# B&R Automation Studio project CombinedLinenSoiledA9KAN (part 7)

#### can_stnCyclic.ab
```automation-basic
PROGRAM _CYCLIC
;----------------------------------------
;Version 1.00 08/02/2005 D.J. First Issue
;----------------------------------------

;The Category, Customer and values from TrackView database are only written every 20 seconds
;unless the database has changed D[65] from TrackView
TimeNow  = clock_ms()
TimeDiff = UINT(TimeNow - TimeLastWrite)
IF (TimeDiff >= 20000) THEN
	WriteEvent 		= TRUE
	TimeLastWrite 	= TimeNow
ELSE IF D[65] <> DatabaseChanged THEN
	WriteEvent 		= TRUE
	TimeLastWrite 	= TimeNow
	DatabaseChanged = D[65]
ENDIF

IF CANOK THEN

	;----------------
	;Set Write values
	;----------------

	;Suction Box 1
	IF Box[1].BagReady THEN
		WriteFrame1021.ControlSignals = BIT_SET(WriteFrame1021.ControlSignals, 1)
	ELSE
		WriteFrame1021.ControlSignals = BIT_CLR(WriteFrame1021.ControlSignals, 1)
	ENDIF

	WriteFrame1101.SP1			= Box[1].SP1
	WriteFrame1101.SP2			= Box[1].SP2
	WriteFrame1101.SP3			= Box[1].SP3
	WriteFrame1101.Category 	= UINT(Box[1].Category)

	WriteFrame1111.Customer 	= Box[1].Customer
	WriteFrame1111.Destination 	= USINT(Box[1].Destination)

	EventWrite1021 = TRUE
	EventWrite1101 = WriteEvent
	EventWrite1111 = WriteEvent
	;Suction Box 1

	;Suction Box 2
	IF Box[2].BagReady THEN
		WriteFrame1022.ControlSignals = BIT_SET(WriteFrame1022.ControlSignals, 1)
	ELSE
		WriteFrame1022.ControlSignals = BIT_CLR(WriteFrame1022.ControlSignals, 1)
	ENDIF

	WriteFrame1102.SP1			= Box[2].SP1
	WriteFrame1102.SP2			= Box[2].SP2
	WriteFrame1102.SP3			= Box[2].SP3
	WriteFrame1102.Category 	= UINT(Box[2].Category)

	WriteFrame1112.Customer 	= Box[2].Customer
	WriteFrame1112.Destination 	= USINT(Box[2].Destination)

	EventWrite1022 = TRUE
	EventWrite1102 = WriteEvent
	EventWrite1112 = WriteEvent
	;Suction Box 2

	;Suction Box 3
	IF Box[3].BagReady THEN
		WriteFrame1023.ControlSignals = BIT_SET(WriteFrame1023.ControlSignals, 1)
	ELSE
		WriteFrame1023.ControlSignals = BIT_CLR(WriteFrame1023.ControlSignals, 1)
	ENDIF

	WriteFrame1103.SP1			= Box[3].SP1
	WriteFrame1103.SP2			= Box[3].SP2
	WriteFrame1103.SP3			= Box[3].SP3
	WriteFrame1103.Category 	= UINT(Box[3].Category)

	WriteFrame1113.Customer 	= Box[3].Customer
	WriteFrame1113.Destination 	= USINT(Box[3].Destination)

	EventWrite1023 = TRUE
	EventWrite1103 = WriteEvent
	EventWrite1113 = WriteEvent
	;Suction Box 3

	;Suction Box 4
	IF Box[4].BagReady THEN
		WriteFrame1024.ControlSignals = BIT_SET(WriteFrame1024.ControlSignals, 1)
	ELSE
		WriteFrame1024.ControlSignals = BIT_CLR(WriteFrame1024.ControlSignals, 1)
	ENDIF

	WriteFrame1104.SP1			= Box[4].SP1
	WriteFrame1104.SP2			= Box[4].SP2
	WriteFrame1104.SP3			= Box[4].SP3
	WriteFrame1104.Category 	= UINT(Box[4].Category)

	WriteFrame1114.Customer 	= Box[4].Customer
	WriteFrame1114.Destination 	= USINT(Box[4].Destination)

	EventWrite1024 = TRUE
	EventWrite1104 = WriteEvent
	EventWrite1114 = WriteEvent
	;Suction Box 4

	;Suction Box 5
	IF Box[5].BagReady THEN
		WriteFrame1025.ControlSignals = BIT_SET(WriteFrame1025.ControlSignals, 1)
	ELSE
		WriteFrame1025.ControlSignals = BIT_CLR(WriteFrame1025.ControlSignals, 1)
	ENDIF

	WriteFrame1105.SP1			= Box[5].SP1
	WriteFrame1105.SP2			= Box[5].SP2
	WriteFrame1105.SP3			= Box[5].SP3
	WriteFrame1105.Category 	= UINT(Box[5].Category)

	WriteFrame1115.Customer 	= Box[5].Customer
	WriteFrame1115.Destination 	= USINT(Box[5].Destination)

	EventWrite1025 = TRUE
	EventWrite1105 = WriteEvent
	EventWrite1115 = WriteEvent
	;Suction Box 5

	;Suction Box 6
	IF Box[6].BagReady THEN
		WriteFrame1026.ControlSignals = BIT_SET(WriteFrame1026.ControlSignals, 1)
	ELSE
		WriteFrame1026.ControlSignals = BIT_CLR(WriteFrame1026.ControlSignals, 1)
	ENDIF

	WriteFrame1106.SP1			= Box[6].SP1
	WriteFrame1106.SP2			= Box[6].SP2
	WriteFrame1106.SP3			= Box[6].SP3
	WriteFrame1106.Category 	= UINT(Box[6].Category)

	WriteFrame1116.Customer 	= Box[6].Customer
	WriteFrame1116.Destination 	= USINT(Box[6].Destination)

	EventWrite1026 = TRUE
	EventWrite1106 = WriteEvent
	EventWrite1116 = WriteEvent
	;Suction Box 6

	;Suction Box 7
	IF Box[7].BagReady THEN
		WriteFrame1027.ControlSignals = BIT_SET(WriteFrame1027.ControlSignals, 1)
	ELSE
		WriteFrame1027.ControlSignals = BIT_CLR(WriteFrame1027.ControlSignals, 1)
	ENDIF

	WriteFrame1107.SP1			= Box[7].SP1
	WriteFrame1107.SP2			= Box[7].SP2
	WriteFrame1107.SP3			= Box[7].SP3
	WriteFrame1107.Category 	= UINT(Box[7].Category)

	WriteFrame1117.Customer 	= Box[7].Customer
	WriteFrame1117.Destination 	= USINT(Box[7].Destination)

	EventWrite1027 = TRUE
	EventWrite1107 = WriteEvent
	EventWrite1117 = WriteEvent
	;Suction Box 7

	;Suction Box 8
	IF Box[8].BagReady THEN
		WriteFrame1028.ControlSignals = BIT_SET(WriteFrame1028.ControlSignals, 1)
	ELSE
		WriteFrame1028.ControlSignals = BIT_CLR(WriteFrame1028.ControlSignals, 1)
	ENDIF

	WriteFrame1108.SP1			= Box[8].SP1
	WriteFrame1108.SP2			= Box[8].SP2
	WriteFrame1108.SP3			= Box[8].SP3
	WriteFrame1108.Category 	= UINT(Box[8].Category)

	WriteFrame1118.Customer 	= Box[8].Customer
	WriteFrame1118.Destination 	= USINT(Box[8].Destination)

	EventWrite1028 = TRUE
	EventWrite1108 = WriteEvent
	EventWrite1118 = WriteEvent
	;Suction Box 8

	;Suction Box 9
	IF Box[9].BagReady THEN
		WriteFrame1029.ControlSignals = BIT_SET(WriteFrame1029.ControlSignals, 1)
	ELSE
		WriteFrame1029.ControlSignals = BIT_CLR(WriteFrame1029.ControlSignals, 1)
	ENDIF

	WriteFrame1109.SP1			= Box[9].SP1
	WriteFrame1109.SP2			= Box[9].SP2
	WriteFrame1109.SP3			= Box[9].SP3
	WriteFrame1109.Category 	= UINT(Box[9].Category)

	WriteFrame1119.Customer 	= Box[9].Customer
	WriteFrame1119.Destination 	= USINT(Box[9].Destination)

	EventWrite1029 = TRUE
	EventWrite1109 = WriteEvent
	EventWrite1119 = WriteEvent
	;Suction Box 9

	;-----------------
	;Service CAN table
	;-----------------

	IF CANdftab_01.status=0 THEN						(*check error level*)
		CANrwtab_01.enable		= 1
		CANrwtab_01.tab_ident	= CANdftab_01.tab_ident (*define tab_id*)
		CANrwtab_01 FUB CANrwtab()						(*initiate CANrwtab*)
		LastError = CANrwtab_01.status
	ENDIF

	;----------------------------------
	;Check for incomming data from CBW1
	;----------------------------------

	;Box 1
	IF EventRead1001 THEN
		EventRead1001 = FALSE
		Box1Cus = UINT(ReadFrame1001.Customer)
	ENDIF

	IF EventRead1011 THEN

		EventRead1011 = FALSE

		Box[1].Live 		= BIT_TST(ReadFrame1011.ControlSignals,0)
		Box[1].LoadFinished = BIT_TST(ReadFrame1011.ControlSignals,1)

		Box[1].Weight		= ReadFrame1011.Weight
		IF (Box1Cus > 0) THEN
			Bag[201].Cus = Box1Cus
		ENDIF
		IF Box[1].Live THEN
			Box[1].LiveTime = 50	;5 seconds
		ENDIF

	ENDIF

;	IF EDGEPOS (Box[1].LoadFinished = 0) THEN
;		Bag[201].Cus = Box1Cus
;	ENDIF
;
;	IF (Bag[201].Cus = 0) THEN
;		Bag[201].Cus = Box1Cus
;	ENDIF

	;Box 2
	IF EventRead1002 THEN
		EventRead1002 = FALSE
		Box2Cus = UINT(ReadFrame1002.Customer)
	ENDIF

	IF EventRead1012 THEN

		EventRead1012 = FALSE

		Box[2].Live 		= BIT_TST(ReadFrame1012.ControlSignals,0)
		Box[2].LoadFinished = BIT_TST(ReadFrame1012.ControlSignals,1)

		Box[2].Weight		= ReadFrame1012.Weight
		IF (Box2Cus > 0) THEN
			Bag[202].Cus = Box2Cus
		ENDIF
		IF Box[2].Live THEN
			Box[2].LiveTime = 50	;5 seconds
		ENDIF

	ENDIF

;	IF EDGEPOS (Box[2].LoadFinished = 0) THEN
;		Bag[202].Cus = Box2Cus
;	ENDIF
;
;	IF (Bag[202].Cus = 0) THEN
;		Bag[202].Cus = Box2Cus
;	ENDIF

	;Box 3
	IF EventRead1003 THEN
		EventRead1003 = FALSE
		Box3Cus = UINT(ReadFrame1003.Customer)
	ENDIF

	IF EventRead1013 THEN

		EventRead1013 = FALSE

		Box[3].Live 		= BIT_TST(ReadFrame1013.ControlSignals,0)
		Box[3].LoadFinished = BIT_TST(ReadFrame1013.ControlSignals,1)

		Box[3].Weight		= ReadFrame1013.Weight
		IF (Box3Cus > 0) THEN
				Bag[203].Cus = Box3Cus
		ENDIF
		IF Box[3].Live THEN
			Box[3].LiveTime = 50	;5 seconds
		ENDIF

	ENDIF

;	IF EDGEPOS (Box[3].LoadFinished = 0) THEN
;		Bag[203].Cus = Box3Cus
;	ENDIF
;
;	IF (Bag[203].Cus = 0) THEN
;		Bag[203].Cus = Box3Cus
;	ENDIF

	;Box 4
	IF EventRead1004 THEN
		EventRead1004 = FALSE
		Box4Cus = UINT(ReadFrame1004.Customer)
	ENDIF

	IF EventRead1014 THEN

		EventRead1014 = FALSE

		Box[4].Live 		= BIT_TST(ReadFrame1014.ControlSignals,0)
		Box[4].LoadFinished = BIT_TST(ReadFrame1014.ControlSignals,1)

		Box[4].Weight		= ReadFrame1014.Weight
		IF (Box4Cus > 0) THEN
			Bag[204].Cus = Box4Cus
		ENDIF
		IF Box[4].Live THEN
			Box[4].LiveTime = 50	;5 seconds
		ENDIF

	ENDIF

;	IF EDGEPOS (Box[4].LoadFinished = 0) THEN
;		Bag[204].Cus = Box4Cus
;	ENDIF
;
;	IF (Bag[204].Cus = 0) THEN
;		Bag[204].Cus = Box4Cus
;	ENDIF

	;Box 5
	IF EventRead1005 THEN
		EventRead1005 = FALSE
		Box5Cus = UINT(ReadFrame1005.Customer)
	ENDIF

	IF EventRead1015 THEN

		EventRead1015 = FALSE

		Box[5].Live 		= BIT_TST(ReadFrame1015.ControlSignals,0)
		Box[5].LoadFinished = BIT_TST(ReadFrame1015.ControlSignals,1)

			Box[5].Weight		= ReadFrame1015.Weight
		IF (Box5Cus > 0) THEN
			Bag[205].Cus = Box5Cus
		ENDIF
		IF Box[5].Live THEN
			Box[5].LiveTime = 50	;5 seconds
		ENDIF

	ENDIF

;	IF EDGEPOS (Box[5].LoadFinished = 0) THEN
;		Bag[205].Cus = Box5Cus
;	ENDIF
;
;	IF (Bag[205].Cus = 0) THEN
;		Bag[205].Cus = Box5Cus
;	ENDIF

	;Box 6
	IF EventRead1006 THEN
		EventRead1006 = FALSE
		Box6Cus = UINT(ReadFrame1006.Customer)
	ENDIF

	IF EventRead1016 THEN

		EventRead1016 = FALSE

		Box[6].Live 		= BIT_TST(ReadFrame1016.ControlSignals,0)
		Box[6].LoadFinished = BIT_TST(ReadFrame1016.ControlSignals,1)

		Box[6].Weight		= ReadFrame1016.Weight
		IF (Box6Cus > 0) THEN
			Bag[206].Cus = Box6Cus
		ENDIF
		IF Box[6].Live THEN
			Box[6].LiveTime = 50	;5 seconds
		ENDIF

	ENDIF

;	IF EDGEPOS (Box[6].LoadFinished = 0) THEN
;		Bag[206].Cus = Box6Cus
;	ENDIF
;
;	IF (Bag[206].Cus = 0) THEN
;		Bag[206].Cus = Box6Cus
;	ENDIF

	;Box 7
	IF EventRead1007 THEN
		EventRead1007 = FALSE
		Dummy = ReadFrame1007.Customer
	ENDIF

	IF EventRead1017 THEN

		EventRead1017 = FALSE

		Box[7].Live 		= BIT_TST(ReadFrame1017.ControlSignals,0)
		Box[7].LoadFinished = BIT_TST(ReadFrame1017.ControlSignals,1)

		Box[7].Weight		= ReadFrame1017.Weight
			IF (ReadFrame1007.Customer > 0) THEN
				Bag[207].Cus = ReadFrame1007.Customer
			ENDIF
		IF Box[7].Live THEN
			Box[7].LiveTime = 50	;5 seconds
		ENDIF

	ENDIF

	;Box 8
	IF EventRead1008 THEN
		EventRead1008 = FALSE
		Dummy = ReadFrame1008.Customer
	ENDIF

	IF EventRead1018 THEN

		EventRead1018 = FALSE

		Box[8].Live 		= BIT_TST(ReadFrame1018.ControlSignals,0)
		Box[8].LoadFinished = BIT_TST(ReadFrame1018.ControlSignals,1)

		Box[8].Weight		= ReadFrame1018.Weight
			IF (ReadFrame1008.Customer > 0) THEN
				Bag[208].Cus = ReadFrame1008.Customer
			ENDIF
		IF Box[8].Live THEN
			Box[8].LiveTime = 50	;5 seconds
		ENDIF

	ENDIF

	;Box 9
	IF EventRead1009 THEN
		EventRead1009 = FALSE
		Dummy = ReadFrame1009.Customer
	ENDIF

	IF EventRead1019 THEN

		EventRead1019 = FALSE

		Box[9].Live 		= BIT_TST(ReadFrame1019.ControlSignals,0)
		Box[9].LoadFinished = BIT_TST(ReadFrame1019.ControlSignals,1)
			Box[9].ReadyToLoad = BIT_TST(ReadFrame1019.ControlSignals,2)
			Box[9].Weight		= ReadFrame1019.Weight
			IF (ReadFrame1009.Customer > 0) THEN
				Bag[209].Cus = ReadFrame1009.Customer
			ENDIF
		IF Box[9].Live THEN
			Box[9].LiveTime = 50	;5 seconds
		ENDIF

	ENDIF

	;-------------------
	;CAN Live / Presence
	;-------------------

	LOOP n = 1 TO 9 DO

		IF (Box[n].LiveTime > 0) THEN
			Box[n].LiveTime = (Box[n].LiveTime - 1)
		ENDIF

		Box[n].Live = (Box[n].LiveTime <> 0)

	ENDLOOP

ENDIF

;Reset Write Event - 20 seconds or Event
WriteEvent = FALSE
END_PROGRAM
```

#### can_stnInit.ab
```automation-basic
PROGRAM _INIT
	(* init program *)

CAN_enable = 1

;BOX 1 Reset CAN data table READ and WRITE events
EventRead1001 	= 0
EventRead1011 	= 0
EventWrite1021 	= 0
EventWrite1101 	= 0
EventWrite1111 	= 0

;BOX 2 Reset CAN data table READ and WRITE events
EventRead1002 	= 0
EventRead1012 	= 0
EventWrite1022 	= 0
EventWrite1102 	= 0
EventWrite1112 	= 0

;BOX 3 Reset CAN data table READ and WRITE events
EventRead1003 	= 0
EventRead1013 	= 0
EventWrite1023 	= 0
EventWrite1103 	= 0
EventWrite1113 	= 0

;BOX 4 Reset CAN data table READ and WRITE events
EventRead1004 	= 0
EventRead1014 	= 0
EventWrite1024 	= 0
EventWrite1104 	= 0
EventWrite1114 	= 0

;BOX 5 Reset CAN data table READ and WRITE events
EventRead1005 	= 0
EventRead1015 	= 0
EventWrite1025 	= 0
EventWrite1105 	= 0
EventWrite1115 	= 0

;BOX 6 Reset CAN data table READ and WRITE events
EventRead1006 	= 0
EventRead1016 	= 0
EventWrite1026 	= 0
EventWrite1106 	= 0
EventWrite1116 	= 0

;BOX 7 Reset CAN data table READ and WRITE events
EventRead1007 	= 0
EventRead1017 	= 0
EventWrite1027 	= 0
EventWrite1107 	= 0
EventWrite1117 	= 0

;BOX 8 Reset CAN data table READ and WRITE events
EventRead1008 	= 0
EventRead1018 	= 0
EventWrite1028 	= 0
EventWrite1108 	= 0
EventWrite1118 	= 0

;BOX 9 Reset CAN data table READ and WRITE events
EventRead1009 	= 0
EventRead1019 	= 0
EventWrite1029 	= 0
EventWrite1109 	= 0
EventWrite1119 	= 0

strcpy(ADR(strName_can_tab), "can_stns")
DOInfo.enable = TRUE
DOInfo.pName  = ADR(strName_can_tab)
DOInfo FUB DatObjInfo()

wTabNum 				= WORD(DOInfo.len / 72)	;Define number of values

CANopen_01.enable		= CAN_enable
CANopen_01.baud_rate	= 25					;Define baud rate - 250 kbit/s
CANopen_01.cob_anz		= wTabNum      			;Define number of link objects
CANopen_01.error_adr	= ADR(error_var)		;Define address for error output
CANopen_01.device		= ADR("SS1.IF1")	    ;Define number of device
CANopen_01.info			= 0

CANopen_01 FUB CANopen()						;Initiate CANopen

IF CANopen_01.status = 0 THEN					;Check error level

	IF (DOInfo.status = 0) THEN

		CANdftab_01.enable			= TRUE
		CANdftab_01.us_ident 		= CANopen_01.us_ident	;Set us_id
		CANdftab_01.table_adr		= DOInfo.pDatObjMem		;Define address of data object
		CANdftab_01.tab_num			= wTabNum

		CANdftab_01 FUB CANdftab()    						;Initiate CANdftab

		IF CANdftab_01.status = 0 THEN
			WriteFrame1021.ControlSignals = BIT_SET(WriteFrame1021.ControlSignals,0);Set Live Signal
			WriteFrame1022.ControlSignals = BIT_SET(WriteFrame1022.ControlSignals,0)
			WriteFrame1023.ControlSignals = BIT_SET(WriteFrame1023.ControlSignals,0)
			WriteFrame1024.ControlSignals = BIT_SET(WriteFrame1024.ControlSignals,0);Set Live Signal
			WriteFrame1025.ControlSignals = BIT_SET(WriteFrame1025.ControlSignals,0)
			WriteFrame1026.ControlSignals = BIT_SET(WriteFrame1026.ControlSignals,0)
			WriteFrame1027.ControlSignals = BIT_SET(WriteFrame1027.ControlSignals,0);Set Live Signal
			WriteFrame1028.ControlSignals = BIT_SET(WriteFrame1028.ControlSignals,0)
			WriteFrame1029.ControlSignals = BIT_SET(WriteFrame1029.ControlSignals,0)
			CANOK = TRUE
		ENDIF

	ENDIF

ENDIF
END_PROGRAM
```

- Data object Logical/Mewa/200ms/CAN/can_stns (Simple, version 1.00.0) - * Suction system (no source held here)

### Program Logical/Mewa/200ms/CAN/can_live (IEC) - * CAN Live status 1-32 to TrackView

#### can_live.ab
```automation-basic
PROGRAM _CYCLIC
(* cyclic program *)

;------------------------------------------
;CAN Live / Status indication to TrackView
;------------------------------------------

;-----------------------------------------
;Revision 1.00 24/11/2005 D.J. First Issue
;-----------------------------------------

;Move CAN Status to Registers

;1-16
CANLive_1.Input[0] = CAN[1].Live
CANLive_1.Input[1] = CAN[2].Live
CANLive_1.Input[2] = CAN[3].Live
CANLive_1.Input[3] = CAN[4].Live
CANLive_1.Input[4] = CAN[5].Live
CANLive_1.Input[5] = CAN[6].Live
CANLive_1.Input[6] = CAN[7].Live
CANLive_1.Input[7] = CAN[8].Live
CANLive_1.Input[8] = CAN[9].Live
CANLive_1.Input[9] = CAN[10].Live
CANLive_1.Input[10] = FALSE ;Box[1].Live
CANLive_1.Input[11] = FALSE ;Box[2].Live
CANLive_1.Input[12] = FALSE ;Box[3].Live
CANLive_1.Input[13] = FALSE ;Box[4].Live
CANLive_1.Input[14] = FALSE ;Box[5].Live
CANLive_1.Input[15] = FALSE ;Box[6].Live

CANLive_1 FUB BIT_ENCODE()

D[76] = CANLive_1.Output

;17-32
CANLive_2.Input[0] = FALSE ;Box[7].Live
CANLive_2.Input[1] = FALSE ;Box[8].Live
CANLive_2.Input[2] = FALSE ;Box[9].Live
CANLive_2.Input[3] = CAN[20].Live
CANLive_2.Input[4] = CAN[21].Live
CANLive_2.Input[5] = CAN[22].Live
CANLive_2.Input[6] = CAN[23].Live
CANLive_2.Input[7] = CAN[24].Live
CANLive_2.Input[8] = CAN[25].Live
CANLive_2.Input[9] = CAN[26].Live
CANLive_2.Input[10] = CAN[27].Live
CANLive_2.Input[11] = CAN[28].Live
CANLive_2.Input[12] = CAN[29].Live
CANLive_2.Input[13] = CAN[30].Live
CANLive_2.Input[14] = CAN[31].Live
CANLive_2.Input[15] = CAN[32].Live

CANLive_2 FUB BIT_ENCODE()

D[77] = CANLive_2.Output
END_PROGRAM
```

### Package Logical/Mewa/KanLink - KanLink Setup tasks

### KanLink.typ - Global data types
```iecst
(********************************************************************
 * COPYRIGHT -- HP
 ********************************************************************
 * Package: KanLink
 * File: KanLink.typ
 * Author: treamsbottom
 * Created: April 23, 2012
 ********************************************************************
 * Data types of package KanLink
 ********************************************************************)

TYPE
	State_typ : 	STRUCT
		Estop : USINT := 1;
		Fault : USINT := 3;
		OK : USINT := 6;
		Warning : USINT := 10;
	END_STRUCT;
	KanLink_Param_typ : 	STRUCT
		Mcn_no : UINT;
		Area : UINT;
		Adr : UINT;
	END_STRUCT;
END_TYPE
```

### KanLink.var - Global variables
```iecst
(********************************************************************
 * COPYRIGHT -- HP
 ********************************************************************
 * Package: KanLink
 * File: KanLink.var
 * Author: treamsbottom
 * Created: April 23, 2012
 ********************************************************************
 * Variables of package KanLink
 ********************************************************************)
VAR
	Batch : ARRAY[0..9] OF BatchData_typ;
	Kan : ARRAY[0..9] OF BatchData_typ;
	PTResp : ARRAY[0..9] OF KL_BTxf_typ;
	PT100 : ARRAY[0..9] OF KL_BTxf_typ;
	McState : State_typ;
END_VAR
VAR RETAIN
	KanLink_Param : ARRAY[0..9] OF KanLink_Param_typ;
END_VAR
```

### Program Logical/Mewa/KanLink/Kan_Drv (IEC) - Empty base sequence

#### Kan_Drv.ab
```automation-basic
;--------------------------------------------
;Sequence Kan_Drv
;--------------------------------------------

PROGRAM _INIT
(* init program *)
END_PROGRAM

PROGRAM _CYCLIC

// Batch Transfer Handshake
//Please enter the index of Kan Bag you want to transfer to the PT+ This was set up in BatchInfo.task
LOOP n = 0 TO (Std.MaxKanLink) DO
;LOOP n = 0 TO 1 DO
	PT100[n].Resp.BatchData = Kan[n];

	ValidCat = 	strcmp(ADR(CAN[n+1].Category), "")
	IF (ValidCat <> 0)THEN
			PT100[n].Resp.xHsDataValid = TRUE;
	ELSE
		PT100[n].Resp.xHsDataValid = FALSE
		PT100[n].Resp.xHsUnloading = FALSE
	ENDIF

	IF CAN[n+1].BagReady THEN
		PT100[n].Resp.xHsReqForUnload = TRUE;
	ELSE
		PT100[n].Resp.xHsReqForUnload = FALSE;
	ENDIF

	CAN[n+1].DropLoad 		= PT100[n].Req.xHreadyForLoad;
	CAN[n+1].LoadDropped  	= PT100[n].Req.xHbatchReceived;
	;CAN[n].Live				= Kanl

		IF CAN[n+1].DropLoad THEN
		PT100[n].Resp.xHsUnloading = TRUE
	ENDIF

	CAN[n+1].Live = IFhlKanLink.Server[n].out.xConnected
	;Status Feedback
	IF Std.HaltSys THEN
		PT100[n].Resp.wState = McState.Estop
	ELSE IF (D[200] > 0) THEN ; alarm present
		PT100[n].Resp.wState = McState.Fault
	ELSE
		PT100[n].Resp.wState = McState.OK
	ENDIF
ENDLOOP
END_PROGRAM
```

#### Kan_Drv.var
```iecst
VAR
	n : UINT;
	ValidCat : DINT;
END_VAR
```

### Program Logical/Mewa/KanLink/zzKanLink (IEC) - KanLink Set up

#### zzKanLinkCyclic.ab - Cyclic code
```automation-basic
(********************************************************************
 * COPYRIGHT -- HP
 ********************************************************************
 * Program: zzKanLink
 * File: zzKanLinkCyclic.ab
 * Author: treamsbottom
 * Created: April 23, 2012
 ********************************************************************
 * Implementation of program zzKanLink
 ********************************************************************)

PROGRAM _CYCLIC
IF NOT init THEN
	KanLink_Param[0].Adr = 12
	KanLink_Param[0].Area = 3
	KanLink_Param[1].Adr = 11
	KanLink_Param[1].Area = 3
	LOOP n = 0 TO (Std.MaxKanLink) DO
	;LOOP n = 0 TO 2 DO
	;Build strings to pass to variable names, only required in a loop as index number changes.
		itoa(n,ADR(sn))	; put n into string
		strcpy(ADR(sReq),"PT100[");build string for variable name (request)
		strcat(ADR(sReq),ADR(sn))
		strcat(ADR(sReq),"].Req")
		strcpy(ADR(sResp),"PT100[");;build string for variable name (response)
		strcat(ADR(sResp),ADR(sn))
		strcat(ADR(sResp),"].Resp")

		IFhlKanLink.Parameter.Server[n].Adr = KanLink_Param[n].Adr ; Populate these arrays .
		IFhlKanLink.Parameter.Server[n].Area = KanLink_Param[n].Area
		IFhlKanLink.Parameter.Server[n].Cmd = 1000 ; cmd from the server are always even
		IFhlKanLink.Parameter.Server[n].CmdOpt = 0
		IFhlKanLink.Parameter.Server[n].TimeOut = 1000 ;ms
		strcpy(ADR(IFhlKanLink.Parameter.Server[n].Name),"PT100") ; Diags Only
		strcpy(ADR(IFhlKanLink.Parameter.Server[n].sReq),ADR(sReq));"zzKanLink:PT100[0].Req")
		strcpy(ADR(IFhlKanLink.Parameter.Server[n].sResp),ADR(sResp));"zzKanLink:PT100[0].Resp")
	ENDLOOP

	;Clean side- Only 1 client for talking to shuttle/driers can be put into a loop as the soiled.
;	IFhlKanLink.Parameter.Client[0].Adr = 15
;	IFhlKanLink.Parameter.Client[0].Area = 3
;	IFhlKanLink.Parameter.Client[0].Cmd = 1000
;	IFhlKanLink.Parameter.Client[0].CmdOpt = 0
;	IFhlKanLink.Parameter.Client[0].CycleTime = 1000;ms
;	strcpy(ADR(IFhlKanLink.Parameter.Client[0].Name),"PTResp")
;	strcpy(ADR(IFhlKanLink.Parameter.Client[0].sReq),"PTResp[0].Req")
;	strcpy(ADR(IFhlKanLink.Parameter.Client[0].sResp),"PTResp[0].Resp")

	IFhlKanLink.in.xRestart = TRUE
	IFmnParam.Out.xParamOK = TRUE
	init = TRUE
	PT100 ; Variable that writes to the PT+
	PTResp ; Variable that reads from PT+ (Clean Side)
ENDIF

END_PROGRAM
```

#### zzKanLinkInit.ab - Initialization code
```automation-basic
(********************************************************************
 * COPYRIGHT -- HP
 ********************************************************************
 * Program: zzKanLink
 * File: zzKanLinkInit.ab
 * Author: treamsbottom
 * Created: April 23, 2012
 ********************************************************************
 * Implementation of program zzKanLink
 ********************************************************************)

PROGRAM _INIT

(* TODO : Add your code here *)

END_PROGRAM
```

#### zzKanLink.var - Local variables
```iecst
(********************************************************************
 * COPYRIGHT -- HP
 ********************************************************************
 * Program: zzKanLink
 * File: zzKanLink.var
 * Author: treamsbottom
 * Created: April 23, 2012
 ********************************************************************
 * Local variables of program zzKanLink
 ********************************************************************)
VAR
	init : BOOL;
	n : UINT;
	sReq : STRING[80];
	sn : STRING[2];
	sResp : STRING[80];
END_VAR
```

### Program Logical/Mewa/KanLink/BatchInfo (IEC) - Empty base sequence

#### BatchInfo.ab
```automation-basic
;--------------------------------------------
;Sequence BatchInfo
;--------------------------------------------

PROGRAM _INIT
(* init program *)
END_PROGRAM

PROGRAM _CYCLIC

	;Please enter Bag number to to send via KannLink Batch info (1002)
	BagNum[0]	= 55
	BagNum[1]	= 60
	BagNum[2]	= 0
	BagNum[3]	= 0
	BagNum[4]	= 0
	BagNum[5]	= 0

	LOOP n = 0 TO Std.MaxKanLink DO
		IF Bag[BagNum[n]].Cat > 0 THEN
			GetTimeStamp.enable = 1
			GetTimeStamp FUB DTGetTime()
			Kan[n].dtTimeStamp = GetTimeStamp.DT1

			;Make a string out of CAT and CUS
			length := itoa(Bag[BagNum[n]].Cat,ADR(myCategoryString));
			length := itoa(Bag[BagNum[n]].Cus,ADR(myCustomerString));
			;strcpy(ADR(myCategoryString),ADR(Bag[BagNum[n]].Cat))
			;strcpy(ADR(myCustomerString),ADR(Bag[BagNum[n]].Cus))

			;copy Bag Data to KanLink Bag data type
			Kan[n].bCntCustomers = 1
			Kan[n].sCategory = myCategoryString
			Kan[n].wTotalWeight = Bag[BagNum[n]].Wgt ;Summaray weight of all Part Customers in the Bag, normally 1
			;Frist Customer in the Bag, allowed for multible Customers in future
			Kan[n].PartBatch[0].sCustomNo = myCustomerString
			Kan[n].PartBatch[0].wCustomWeight = Bag[BagNum[n]].Wgt
		ELSE
			strcpy(ADR(myCategoryString),ADR(""));
			strcpy(ADR(myCustomerString),ADR(""));
			Kan[n].bCntCustomers = 0
			Kan[n].sCategory = myCategoryString
			Kan[n].wTotalWeight = 0 ;Summaray weight of all Part Customers in the Bag, normally 1
			;Frist Customer in the Bag, allowed for multible Customers in future
			Kan[n].PartBatch[0].sCustomNo = myCustomerString
			Kan[n].PartBatch[0].wCustomWeight = 0
		ENDIF
		Batch[n] = Kan[n] ; Populate array for PT+ PVI
	ENDLOOP
;
;	//Batch info for all Batches
;	Bel_1_BI.Resp.BatchData[0] = Kan[0];
;	Bel_1_BI.Resp.BatchData[1] = Kan[0];
;	Bel_1_BI.Resp.BatchData[2] = Kan[0];
;	Bel_1_BI.Resp.BatchData[3] = Kan[0];
;	Bel_1_BI.Resp.BatchData[4] = Kan[0];
;	Bel_1_BI.Resp.BatchData[5] = Kan[0];
;
;
;	IF (Bel_1_BI.Req.wCntPositions >= 0) THEN
;		n = Bel_1_BI.Req.wCntPositions;
;		Bel_1_BI.Resp.wCntPositions =  Bel_1_BI.Req.wCntPositions;
;		IF (n = 0) OR (n >= 1) THEN
;			Bel_1_BI.Resp.wNoOfPositions[0] = Bel_1_BI.Req.wNoOfPosition[0];
;			Bel_1_BI.Resp.BatchData[0] = Kan[Bel_1_BI.Req.wNoOfPosition[0]];
;		ENDIF
;		IF (n = 0) OR (n >= 2) THEN
;			Bel_1_BI.Resp.wNoOfPositions[1] = Bel_1_BI.Req.wNoOfPosition[1];
;			Bel_1_BI.Resp.BatchData[1] = Kan[Bel_1_BI.Req.wNoOfPosition[1]];
;		ENDIF
;		IF (n = 0) OR (n >= 3) THEN
;			Bel_1_BI.Resp.wNoOfPositions[2] = Bel_1_BI.Req.wNoOfPosition[2];
;			Bel_1_BI.Resp.BatchData[2] = Kan[Bel_1_BI.Req.wNoOfPosition[2]];
;		ENDIF
;		IF (n = 0) OR (n >= 4) THEN
;			Bel_1_BI.Resp.wNoOfPositions[3] = Bel_1_BI.Req.wNoOfPosition[3];
;			Bel_1_BI.Resp.BatchData[3] = Kan[Bel_1_BI.Req.wNoOfPosition[3]];
;		ENDIF
;		IF (n = 0) OR (n >= 5) THEN
;			Bel_1_BI.Resp.wNoOfPositions[4] = Bel_1_BI.Req.wNoOfPosition[4];
;			Bel_1_BI.Resp.BatchData[4] = Kan[Bel_1_BI.Req.wNoOfPosition[4]];
;		ENDIF
;		IF (n = 0) OR (n = 6) THEN
;			Bel_1_BI.Resp.wNoOfPositions[5] = Bel_1_BI.Req.wNoOfPosition[5];
;			Bel_1_BI.Resp.BatchData[5] = Kan[Bel_1_BI.Req.wNoOfPosition[5]];
;		ENDIF
;	ENDIF
;
;
;
END_PROGRAM
```

#### BatchInfo.var
```iecst
VAR
	BagNum : ARRAY[0..10] OF UINT;
	n : UINT;
	length : UINT;
	myCategoryString : STRING[11];
	myCustomerString : STRING[11];
	nxt_adr : UDINT;
	GetTimeStamp : DTGetTime;
END_VAR
```

### Package Logical/Mewa/KGFramework - Standard-Packages

### Package Logical/Mewa/KGFramework/Pkg_KGStandard - Kannegiesser Standards

### kgMachineState.var - Package variables
```iecst
(********************************************************************
 * COPYRIGHT -- Herbert Kannegiesser GmbH
 ********************************************************************
 * Package: Pkg_KGStandard
 * File: kgMachineState.var
 * Author: hunholz
 * Created: January 27, 2012
 ********************************************************************
 * Variables of package Pkg_KGStandard
 ********************************************************************)
VAR CONSTANT
	KG_MACHINESTATE_OFF : UINT := 0; (*Machine is turned off*)
	KG_MACHINESTATE_EMERGENCYSTOP : UINT := 1; (*Emergency stop*)
	KG_MACHINESTATE_SAFESTOP : UINT := 2; (*Safe stop*)
	KG_MACHINESTATE_FAULT : UINT := 3; (*Fault*)
	KG_MACHINESTATE_FAULT_GONE : UINT := 4; (*Fault, wait for acknowledge*)
	KG_MACHINESTATE_SERVICE : UINT := 5; (*Service*)
	KG_MACHINESTATE_AUTOMATIC_RUN : UINT := 6; (*Automatic Run*)
	KG_MACHINESTATE_STOP : UINT := 7; (*Stop*)
	KG_MACHINESTATE_WAIT_AUTOMATIC : UINT := 8; (*Automatic Wait (Standby)*)
	KG_MACHINESTATE_WAIT_MAN : UINT := 9; (*Automatic Wait for manual action*)
	KG_MACHINESTATE_WARNING : UINT := 10; (*Automatic Warning*)
END_VAR
(*Special states for dryer*)
VAR CONSTANT
	KG_MACHINESTATE_DRY_HEATING : UINT := 30; (*Automatic heating*)
	KG_MACHINESTATE_DRY_COOLDOWN : UINT := 31; (*Automatic cooldown*)
	KG_MACHINESTATE_DRY_CLEAN_FILTER : UINT := 32; (*Automatic clean filter*)
	KG_MACHINESTATE_DRY_AFTERRUN : UINT := 33; (*Automatic afterrun*)
	KG_MACHINESTATE_DRY_FAN_CLEAN : UINT := 34; (*Automatic running cleaning fan*)
END_VAR
(*Special states for conveyor*)
VAR CONSTANT
	KG_MACHINESTATE_CONV_FWD : UINT := 40; (*Automatic running forward*)
	KG_MACHINESTATE_CONV_FWD2 : UINT := 41; (*Automatic running forward 2nd speed*)
	KG_MACHINESTATE_CONV_REV : UINT := 42; (*Automatic running reverse*)
	KG_MACHINESTATE_CONV_REV2 : UINT := 43; (*Automatic running reverse 2nd speed*)
END_VAR
```

### Library Logical/Mewa/KGFramework/Pkg_KGStandard/KGstdLib (IEC) - Kannegiesser Hilfsfunktionen
Depends on: astime, AsIODiag, Ethernet, AsBrStr, DataObj, AsArLog

#### KGstdLib.var - Exported constants
```iecst
(********************************************************************
 * COPYRIGHT -- Microsoft
 ********************************************************************
 * Library: KGstd
 * File: KGstd.var
 * Author: hunholz
 * Created: June 23, 2011
 ********************************************************************
 * Constants of library KGstd
 ********************************************************************)
VAR CONSTANT
	KG_ERR_RB_NOREAD : UINT := 1;
	KG_ERR_RB_POINTER : UINT := 2;
	KG_ERR_RB_WRITEPOINTER : UINT := 3;
	KG_ERR_RB_READPOINTER : UINT := 4;
	KG_ERR_RB_STARTPOINTER : UINT := 5;
	KG_ERR_RB_LOCPOINTER : UINT := 6;
	KG_ERR_RB_SIZE : UINT := 7;
	KG_ERR_GETETHPORT_IFSTRING : UINT := 21;
	KG_ERR_GETETHPORT_ADRIF : UINT := 22;
	KG_ERR_WRONGSIZES : UINT := 30;
	KG_INFO_DO_NEW : UINT := 31;
	KG_ERR_NULPOINTER : UINT := 40;
	KG_ERR_NULLSTRING : UINT := 41;
END_VAR
(*RB Modus für kgRBloc*)
VAR CONSTANT
	KG_RB_LOC_MODE_ABSOLUTE : USINT := 0;
	KG_RB_LOC_MODE_FROMSTART : USINT := 1;
	KG_RB_LOC_MODE_FROMEND : USINT := 2;
END_VAR
(*CPU Identifier*)
VAR CONSTANT
	KG_CPU_X20CP3484 : UDINT := 16#23A6;
	KG_CPU_X20CP1484 : UDINT := 16#23A5;
	KG_CPU_X20CP1484_1 : UDINT := 16#AABE;
	KG_CPU_X20CP3484_1 : UDINT := 16#AABF;
	KG_CPU_X20CP1486 : UDINT := 16#2164;
	KG_CPU_X20CP3486 : UDINT := 16#1F19;
	KG_CPU_X20CP3585 : UDINT := 16#C3AF;
	KG_CPU_PP420_1043_75 : UDINT := 16#23BD;
	KG_CPU_PP65_0571_P74 : UDINT := 16#A964;
	KG_CPU_CTT_11 : UDINT := 16#A2BC;
	KG_CPU_PCT_03 : UDINT := 16#A7DD;
	KG_CPU_PCT_04 : UDINT := 16#B399;
END_VAR
(*Units*)
VAR CONSTANT
	KG_UNIT_METRIC : USINT := 0;
	KG_UNIT_US : USINT := 1;
END_VAR
```

#### KGstdLib.fun - Exported functions and function blocks
```iecst
(********************************************************************
 * COPYRIGHT -- Microsoft
 ********************************************************************
 * Library: KGstd
 * File: KGstd.fun
 * Author: hunholz
 * Created: June 23, 2011
 ********************************************************************
 * Functions and function blocks of library KGstd
 ********************************************************************)

FUNCTION_BLOCK kgGetEthPort (*Returns the CPUs ethernet port as string*)
	VAR_INPUT
		enable : BOOL;
		adrIF : UDINT;
	END_VAR
	VAR_OUTPUT
		status : UINT;
	END_VAR
	VAR
		_bStep : USINT;
		DiagCreateInfo_CPU : DiagCreateInfo;
		DiagGetNumInfo_CPU : DiagGetNumInfo;
		DiagDisposeInfo_CPU : DiagDisposeInfo;
		_xReady : BOOL;
	END_VAR
END_FUNCTION_BLOCK

FUNCTION kgitoa_udint : UINT (*Wandelt UDINT Werte in einen String*)
	VAR_INPUT
		num : UDINT;
	END_VAR
	VAR_IN_OUT
		str : STRING[11];
	END_VAR
	VAR
		_num : UDINT;
		_digit : UDINT;
		_sdigit : STRING[1];
		_bdigit : REFERENCE TO USINT;
	END_VAR
END_FUNCTION

FUNCTION kgatoi_udint : UINT (*String in UDINT wandeln*)
	VAR_INPUT
		str : STRING[11];
	END_VAR
	VAR_IN_OUT
		num : UDINT;
	END_VAR
	VAR
		_len : UINT;
		_result : UINT;
		_sdigit : STRING[1];
		_bdigit : REFERENCE TO USINT;
		_mul : UDINT;
		_digit : UDINT;
		_i : INT;
	END_VAR
END_FUNCTION

FUNCTION kgatoi_uint : UINT (*atoi für UINT mit Fehlermeldung*)
	VAR_INPUT
		str : STRING[11];
	END_VAR
	VAR_IN_OUT
		num : UINT;
	END_VAR
	VAR
		_result : UINT;
		_len : INT;
		_sdigit : STRING[1];
		_bdigit : REFERENCE TO USINT;
		_mul : UINT;
		_i : INT;
		_digit : USINT;
	END_VAR
END_FUNCTION

FUNCTION_BLOCK kgNextBatchNoLong (*Generiert eine neue Postennummer*)
	VAR_INPUT
		Enable : BOOL; (*Positive Flanke erzeugt neue Nummer*)
		Group : USINT; (*0..7*)
	END_VAR
	VAR_OUTPUT
		Status : UINT; (*0 : OK, 1 : Maximale Anzahl möglicher Nummern pro Tag erreich, B&R Werte*)
		BatchNo : UDINT;
	END_VAR
	VAR
		_bOldYear : USINT;
		_bOldMonth : USINT;
		_bOldDay : USINT;
		DTStrucGetTime : DTStructureGetTime;
		_dtStruc : DTStructure;
		_bGroup : USINT;
		_wNo : UINT;
		_bStep : USINT;
		_diBatchNo : DatObjInfo;
		_pBatchNo : REFERENCE TO UDINT;
		_dwBatchNo : DatObjWrite;
		_dcBatchNo : DatObjCreate;
		zzEdge00000 : BOOL;
	END_VAR
END_FUNCTION_BLOCK

FUNCTION_BLOCK kgGetMacAdress (*Nur im Init-Up aufrufen*)
	VAR_INPUT
		Enable : BOOL;
	END_VAR
	VAR_OUTPUT
		Mac : MAC_type;
		Status : UINT;
	END_VAR
	VAR
		_gep : kgGetEthPort;
		_sIF : STRING[23];
		_exi : ETHxinfo;
		_bMAC : MAC_type;
	END_VAR
END_FUNCTION_BLOCK

FUNCTION_BLOCK kgGetBatchNoUnique (*Batchnummer als Unique Identifier 16 Byte*)
	VAR_INPUT
		Enable : BOOL;
		Mac : MAC_type;
	END_VAR
	VAR_OUTPUT
		BatchNo : GUID_type;
		Status : UINT;
	END_VAR
	VAR
		DTGetTime_0 : DTGetTime;
		_time : TIME;
	END_VAR
END_FUNCTION_BLOCK

FUNCTION kgBatchNoToUDINT : UDINT (*Extrahiere aus GUID ein UDINT*)
	VAR_INPUT
		GUID : GUID_type;
	END_VAR
	VAR
		_udint : REFERENCE TO UDINT;
	END_VAR
END_FUNCTION

FUNCTION_BLOCK kgUSINT16toGUID (*Konvertiere USINT-Array to GUID_typ*)
	VAR_INPUT
		usintarray : ARRAY[0..15] OF USINT;
	END_VAR
	VAR_OUTPUT
		GUID : GUID_type;
	END_VAR
END_FUNCTION_BLOCK

FUNCTION_BLOCK kgGUIDtoSTRING (*GUID-String erzeugen*)
	VAR_INPUT
		GUID : GUID_type;
	END_VAR
	VAR_OUTPUT
		sOut : STRING[36];
	END_VAR
	VAR
		usintarray : REFERENCE TO ARRAY[0..15] OF USINT;
		_StringArray : REFERENCE TO ARRAY[0..36] OF USINT;
		_Ptr : INT;
		_i : INT;
		_b : USINT;
	END_VAR
END_FUNCTION_BLOCK

FUNCTION_BLOCK kgLogLine (*Logzeile mit zwei numerischen Variablen erzeugen*)
	VAR_INPUT
		sLoglineTemplate : STRING[127];
		lAttr1 : UDINT;
		lAttr2 : UDINT;
	END_VAR
	VAR_OUTPUT
		sLogline : STRING[127];
		pLogline : UDINT;
	END_VAR
	VAR
		_iPos1 : INT;
		_iPos2 : INT;
		_iCrs : INT;
		sValue : STRING[11];
		_sTemp : STRING[127];
	END_VAR
END_FUNCTION_BLOCK

FUNCTION_BLOCK kgArLogWrite (*Checks ident on > 0 and formats string with two numbers*)
	VAR_INPUT
		enable : BOOL;
		ident : UDINT;
		logLevel : UDINT;
		errornr : UDINT;
		text : STRING[127];
		var1 : UDINT;
		var2 : UDINT;
	END_VAR
	VAR_OUTPUT
		status : UINT;
	END_VAR
	VAR
		_AsArLogWrite : AsArLogWrite;
		_kgLogLine : kgLogLine;
	END_VAR
END_FUNCTION_BLOCK

FUNCTION_BLOCK kgRBinsert (*Insert any entry into a ringbuffer*)
	VAR_INPUT
		pEntry : UDINT;
		lLenEntry : UDINT;
		doIdent : UDINT;
		doLen : UDINT;
	END_VAR
	VAR_OUTPUT
		wStatus : UINT;
	END_VAR
	VAR_IN_OUT
		wPtrStart : UINT;
		wPtrWrite : UINT;
		wPtrRead : UINT;
	END_VAR
	VAR
		doWrite : DatObjWrite;
		_lRBlen : UDINT;
		_wPtrMax : UINT;
	END_VAR
END_FUNCTION_BLOCK

FUNCTION_BLOCK kgRBread (*Reads one entry and moves the readpointer*)
	VAR_INPUT
		pEntry : UDINT;
		lLenEntry : UDINT;
		doIdent : UDINT;
		doLen : UDINT;
		wPtrStart : UINT;
		wPtrWrite : UINT;
	END_VAR
	VAR_OUTPUT
		wStatus : UINT;
	END_VAR
	VAR_IN_OUT
		wPtrRead : UINT;
	END_VAR
	VAR
		doRead : DatObjRead;
		_lRBlen : UDINT;
		_wPtrMax : UINT;
	END_VAR
END_FUNCTION_BLOCK

FUNCTION_BLOCK kgRBloc (*Free Readpointer access*)
	VAR_INPUT
		pEntry : UDINT;
		lLenEntry : UDINT;
		doIdent : UDINT;
		doLen : UDINT;
		wPtrStart : UINT;
		wPtrWrite : UINT;
		wPtrLoc : UINT;
		bMode : USINT; (*Lese relativ zum Start- oder Schreibzeiger*)
	END_VAR
	VAR_OUTPUT
		wStatus : UINT;
	END_VAR
	VAR
		doRead : DatObjRead;
		_lRBlen : UDINT;
		_wPtrMax : UINT;
		_wPtrLoc : UINT;
		_wActLen : UINT;
	END_VAR
END_FUNCTION_BLOCK

FUNCTION kgGUIDisZero : BOOL (*Prüfen, ob alle 16 Byte der GUID 0 sind.*)
	VAR_INPUT
		GUID : GUID_type;
	END_VAR
	VAR
		_bGUID : REFERENCE TO ARRAY[0..15] OF USINT;
		_i : USINT;
	END_VAR
END_FUNCTION

FUNCTION_BLOCK kgRBcreate (*Erzeuge Datenobjekt für Ringbuffer*)
	VAR_INPUT
		sName : STRING[10]; (*Name des Datenobjekts*)
		bMemType : USINT; (*Speichertyp*)
		wCntEntry : UINT; (*Mindestanzahl der RB_Einträge*)
		lLenEntry : UDINT; (*Länge des einzelnen Eintrags*)
	END_VAR
	VAR_OUTPUT
		doIdent : UDINT; (*Identifier des Datenobjekts*)
		doLen : UDINT; (*Länge des Datenobjekts*)
		wStatus : UINT; (*Status*)
		pDatObjMem : UDINT;
	END_VAR
	VAR_IN_OUT
		wPtrWrite : UINT; (*Schreibzeiger*)
		wPtrRead : UINT; (*Lesezeiger*)
		wPtrStart : UINT; (*Startzeiger*)
	END_VAR
	VAR
		_diRB : DatObjInfo;
		_dcRB : DatObjCreate;
		_ddRB : DatObjDelete;
	END_VAR
END_FUNCTION_BLOCK

FUNCTION_BLOCK kgRBbulkloc (*Lese mehrere Einträge gleichzeitig in ein Array*)
	VAR_INPUT
		pEntry : UDINT; (*Zeiger auf den Zielbereich*)
		lLenEntry : UDINT; (*Länge eines Eintrags*)
		wCntEntry : UINT; (*Anzahl Einträge*)
		doIdent : UDINT;
		doLen : UDINT;
		wPtrStart : UINT;
		wPtrWrite : UINT;
		wPtrLoc : UINT;
		bMode : USINT;
	END_VAR
	VAR_OUTPUT
		wStatus : UINT;
		wCntLoc : UINT;
	END_VAR
	VAR
		_lRBlen : UDINT;
		_wPtrMax : UINT;
		_wActLen : UINT;
		_wPtrLoc : UINT;
		_i : UINT;
		_doRead : DatObjRead;
	END_VAR
END_FUNCTION_BLOCK

FUNCTION kgGetLineNumberW3 : USINT (*Maschinennummer und -typ aus Stationsadresse berechnen*)
	VAR_INPUT
		Station : USINT;
		pMachineType : UDINT;
	END_VAR
	VAR
		_MachineType : REFERENCE TO kgMachinetypeW3_typ;
	END_VAR
END_FUNCTION

FUNCTION_BLOCK kgInitBatchNoLong (*Legt ggf. Datenobjekt zum Speichern der laufenden Postennummer an*)
	VAR_INPUT
		Enable : BOOL;
	END_VAR
	VAR_OUTPUT
		Status : UINT;
	END_VAR
	VAR
		_bStep : USINT;
		_diBatchNo : DatObjInfo;
		_dcBatchNo : DatObjCreate;
		_BatchNo : UDINT;
	END_VAR
END_FUNCTION_BLOCK

FUNCTION kgGetMachineAdressW3 : USINT (*Ermittelt die Maschinenadresse aus Liniennummer und Maschinentyp*)
	VAR_INPUT
		LineNumber : USINT;
		MachineType : kgMachinetypeW3_typ;
	END_VAR
	VAR
		_diMachineType : REFERENCE TO DINT;
	END_VAR
END_FUNCTION

FUNCTION_BLOCK kgCheckDo (*Prüfe auf Datenobjekt und erzeuge es ggf. neu*)
	VAR_INPUT
		Enable : BOOL;
		pName : UDINT;
		MinLen : UDINT;
		NomLen : UDINT;
		Create : BOOL;
		MemType : USINT;
	END_VAR
	VAR_OUTPUT
		doId : UDINT;
		doMem : UDINT;
		doLen : UDINT;
		Status : UINT;
	END_VAR
	VAR
		_wStep : UINT;
		_doInfo : DatObjInfo;
		_xReady : BOOL;
		_doDelete : DatObjDelete;
		_doCreate : DatObjCreate;
	END_VAR
END_FUNCTION_BLOCK

FUNCTION kgXOR : USINT (*XOR über Byte-Feld*)
	VAR_INPUT
		pMem : UDINT; (*Speicher*)
		wLen : UINT; (*Länge*)
		bInit : USINT; (*Startwert*)
		pStatus : UDINT; (*Status*)
		pWordResult : UDINT;
	END_VAR
	VAR
		_wDynStatus : REFERENCE TO UINT;
		_xStatusOk : BOOL;
		_bMem : REFERENCE TO ARRAY[1..65535] OF USINT;
		_xWordResultOk : BOOL;
		_bWordResult : REFERENCE TO ARRAY[0..1] OF USINT;
		_i : UINT;
	END_VAR
END_FUNCTION

FUNCTION kgUnitconfREALtoDisplay : REAL (*Wandelt Wert entsprechend der Unit*)
	VAR_INPUT
		Value : REAL;
		Unit : UINT;
		LocUnit : USINT;
		pDigits : UDINT;
		pUnit : UDINT;
	END_VAR
	VAR
		lDigits : UDINT;
		sUnit : STRING[11];
	END_VAR
END_FUNCTION

FUNCTION kgUnitconfDisplayToREAL : REAL (*Wandelt Wert entsprechend der Unit*)
	VAR_INPUT
		Display : REAL;
		Unit : UINT;
		LocUnit : USINT;
	END_VAR
END_FUNCTION

FUNCTION kgGetProgdata : UINT (*Read Programdata from a dataobject*)
	VAR_INPUT
		sBaseName : STRING[11];
		wProgNo : UINT;
		wProgMaxNo : UINT;
		pMem : UDINT;
		lSize : UDINT;
	END_VAR
	VAR
		_sIndex : STRING[5];
		_sIndex1 : STRING[5];
		_sName : STRING[16];
		_diProg : DatObjInfo;
	END_VAR
END_FUNCTION
```

#### kgGetEthPort.st - Returns the CPUs ethernet port as string
```iecst
(********************************************************************
 * COPYRIGHT -- Microsoft
 ********************************************************************
 * Library: Netlink
 * File: GetEthPort.st
 * Author: hunholz
 * Created: June 30, 2011
 ********************************************************************
 * Implementation of library Netlink
 ********************************************************************)

(* Returns the CPUs ethernet port as string *)
FUNCTION_BLOCK kgGetEthPort

	IF enable THEN

		IF adrIF <= 16#3FFF THEN

			_bStep := 10;
			status := KG_ERR_GETETHPORT_ADRIF;
			RETURN;

		END_IF

		_xReady := FALSE;

		REPEAT

			CASE (_bStep) OF

				10:
				// Create Info
					DiagCreateInfo_CPU(enable := TRUE, infoKind := asdiagPLUGGED);

					status := DiagCreateInfo_CPU.status;

					IF (status = ERR_OK) THEN
			  			_bStep := 12;
					END_IF;

				12:
					// Get Info
					DiagGetNumInfo_CPU(enable := TRUE,
											ident := DiagCreateInfo_CPU.ident,
											index := 0,
											infoCode := asdiagPLUGGED_MODNO);

					status := DiagGetNumInfo_CPU.status;

					IF (status = ERR_OK) THEN

						CASE DiagGetNumInfo_CPU.value OF

							KG_CPU_X20CP1484, KG_CPU_X20CP1484_1, KG_CPU_X20CP3484_1, KG_CPU_X20CP1486, KG_CPU_X20CP3486, KG_CPU_X20CP3585, KG_CPU_X20CP3484 :
								brsstrcpy(adrIF, ADR('IF2'));

							KG_CPU_PP420_1043_75, KG_CPU_CTT_11, KG_CPU_PP65_0571_P74, KG_CPU_PCT_04, KG_CPU_PCT_03:
								brsstrcpy(adrIF, ADR('IF5'));

							ELSE	// keinen gültigen B&R ID-Code gefunden
								brsstrcpy(adrIF, ADR('ERR'));
								status := KG_ERR_GETETHPORT_IFSTRING;

						END_CASE

						_bStep := 14;

					ELSIF (status <> ERR_FUB_BUSY) THEN
						_bStep := 10;
					END_IF;

				14:
					// Write string to variable

					DiagDisposeInfo_CPU(enable := TRUE, ident := DiagCreateInfo_CPU.ident);

					status := DiagDisposeInfo_CPU.status;

					_xReady := (status = ERR_OK);

					IF (status <> ERR_FUB_BUSY) THEN

						_bStep := 10;
						DiagCreateInfo_CPU(enable := FALSE);
						DiagDisposeInfo_CPU(enable := FALSE);
						DiagGetNumInfo_CPU(enable := FALSE);

					END_IF;

				ELSE

					_bStep := 10;
					status := ERR_FUB_BUSY;

			END_CASE;

			UNTIL

			status <> ERR_OK OR _xReady

		END_REPEAT

	ELSE

		status := ERR_FUB_ENABLE_FALSE;
		_bStep := 10;

	END_IF

END_FUNCTION_BLOCK
```

#### kgUnitconfREALtoDisplay.st - Wandelt Wert entsprechend der Unit
```iecst
(********************************************************************
 * COPYRIGHT -- Herbert Kannegiesser GmbH
 ********************************************************************
 * Library: KGstdLib
 * File: kgUnitconfREALtoDisplay.st
 * Author: hunholz
 * Created: March 15, 2012
 ********************************************************************
 * Implementation of library KGstdLib
 ********************************************************************)

(* Wandelt Wert entsprechend der Unit *)
FUNCTION kgUnitconfREALtoDisplay

	lDigits := 0;
	sUnit := '';

	CASE Unit OF

		2,60,70,80,901:

			// 1/10
			kgUnitconfREALtoDisplay := Value * 0.1;
			lDigits := 1;

			CASE Unit OF

				2:
					// Sekunden
					sUnit := 's';

				60:
					// Hertz
					sUnit := 'Hz';

				70:
					// Winkel
					sUnit := '°';

				80:
					// Prozent
					sUnit := '%';

			END_CASE

		90,902:
			// 1/100
			kgUnitconfREALtoDisplay := Value * 0.01;
			lDigits := 2;

			CASE Unit OF

				90:
					// g
					sUnit := 'g';

			END_CASE

		4,903:

			// 1/1000
			kgUnitconfREALtoDisplay := Value * 0.001;
			lDigits := 3;

			CASE Unit OF

				4:
					// Sekunde
					sUnit := 's';

			END_CASE

		10:
			// liter Gallonen
			IF LocUnit = KG_UNIT_US THEN
				kgUnitconfREALtoDisplay := Value * 0.2641721;
				lDigits := 1;
				sUnit := 'US gal';
			ELSE
				kgUnitconfREALtoDisplay := Value;
				sUnit := 'l';
			END_IF

		11:
			// milliliter Ounce
			IF LocUnit = KG_UNIT_US THEN
				kgUnitconfREALtoDisplay := Value * 0.03381402;
				lDigits := 3;
				sUnit := 'fl.Oz.';

			ELSE
				kgUnitconfREALtoDisplay := Value;
				sUnit := 'ml';
			END_IF

		20:
			// mm inch
			IF LocUnit = KG_UNIT_US THEN
				kgUnitconfREALtoDisplay := Value * 0.03937;
				lDigits := 2;
				sUnit := 'inch';
			ELSE
				kgUnitconfREALtoDisplay := Value;
				sUnit := 'mm';
			END_IF

		21:
			// mm cm inch
			IF LocUnit = KG_UNIT_US THEN
				kgUnitconfREALtoDisplay := Value * 0.03937;
				lDigits := 2;
				sUnit := 'inch';
			ELSE
				kgUnitconfREALtoDisplay := Value * 0.1;
				lDigits := 1;
				sUnit := 'cm';
			END_IF

		22:
			// mm dm inch
			IF LocUnit = KG_UNIT_US THEN
				kgUnitconfREALtoDisplay := Value * 0.03937;
				sUnit := 'inch';
			ELSE
				kgUnitconfREALtoDisplay := Value * 0.01;
				sUnit := 'dm';
			END_IF
			lDigits := 2;

		23:
			// mm m feet
			IF LocUnit = KG_UNIT_US THEN
				kgUnitconfREALtoDisplay := Value * 0.00328;
				sUnit := 'ft';
			ELSE
				kgUnitconfREALtoDisplay := Value * 0.001;
				sUnit := 'm';
			END_IF
			lDigits := 3;

		30:
			// 0,1kg kg lbs
			IF LocUnit = KG_UNIT_US THEN
				kgUnitconfREALtoDisplay := Value * 0.220462;
				sUnit := 'lbs';
			ELSE
				kgUnitconfREALtoDisplay := Value * 0.1;
				sUnit := 'kg';
			END_IF
			lDigits := 1;

		40:
			// 0,1 °C °C °F
			IF LocUnit = KG_UNIT_US THEN
				kgUnitconfREALtoDisplay := (Value * 0.18) + 32.0;
				sUnit := '°F';
			ELSE
				kgUnitconfREALtoDisplay := Value * 0.1;
				sUnit := '°C';
			END_IF
			lDigits := 1;

		41:
			// °C °C °F
			IF LocUnit = KG_UNIT_US THEN
				kgUnitconfREALtoDisplay := (Value * 1.8) + 32.0;
				sUnit := '°F';
			ELSE
				kgUnitconfREALtoDisplay := Value;
				sUnit := '°C';
			END_IF

		50:
			// 0,1 bar bar psi
			IF LocUnit = KG_UNIT_US THEN
				kgUnitconfREALtoDisplay := Value * 1.450368;
				sUnit := 'psi';
			ELSE
				kgUnitconfREALtoDisplay := Value * 0.1;
				lDigits := 1;
				sUnit := 'bar';
			END_IF

		310:
			// 0,01 l/kg l/kg gal/lbs
			IF LocUnit = KG_UNIT_US THEN
				kgUnitconfREALtoDisplay := Value * 0.00119827;
				lDigits := 2;
				sUnit := 'gal/lbs';
			ELSE
				kgUnitconfREALtoDisplay := Value * 0.01;
				lDigits := 1;
				sUnit := 'l/kg';
			END_IF

		ELSE

			kgUnitconfREALtoDisplay := Value;

			CASE Unit OF

				1:
					sUnit := 's';
				3:
					sUnit := 'min';
				81:
					sUnit := '%';

			END_CASE

	END_CASE

	IF pDigits > 0 THEN

		brsmemcpy(pDigits, ADR(lDigits), SIZEOF(lDigits));

	END_IF

	IF pUnit > 0 THEN

		brsmemcpy(pUnit, ADR(sUnit), SIZEOF(sUnit));

	END_IF

END_FUNCTION
```

#### kgUnitconfDisplayToREAL.st - Wandelt Wert entsprechend der Unit
```iecst
(********************************************************************
 * COPYRIGHT -- Herbert Kannegiesser GmbH
 ********************************************************************
 * Library: KGstdLib
 * File: kgUnitconfDisplayToREAL.st
 * Author: hunholz
 * Created: March 15, 2012
 ********************************************************************
 * Implementation of library KGstdLib
 ********************************************************************)

(* Wandelt Wert entsprechend der Unit *)
FUNCTION kgUnitconfDisplayToREAL

	CASE Unit OF

		2,60,70,80,901:
			// 1/10
			kgUnitconfDisplayToREAL := Display * 10;

		90,902:
			// 1/100
			kgUnitconfDisplayToREAL := Display * 100;

		4,903:
			// 1/1000
			kgUnitconfDisplayToREAL := Display * 1000;

		10:
			// liter Gallonen
			IF LocUnit = KG_UNIT_US THEN
				kgUnitconfDisplayToREAL := Display / 0.2641721;
			ELSE
				kgUnitconfDisplayToREAL := Display;
			END_IF

		11:
			// milliliter Ounce
			IF LocUnit = KG_UNIT_US THEN
				kgUnitconfDisplayToREAL := Display / 0.03381402;
			ELSE
				kgUnitconfDisplayToREAL := Display;
			END_IF

		20:
			// mm inch
			IF LocUnit = KG_UNIT_US THEN
				kgUnitconfDisplayToREAL := Display / 0.03937;
			ELSE
				kgUnitconfDisplayToREAL := Display;
			END_IF

		21:
			// mm cm inch
			IF LocUnit = KG_UNIT_US THEN
				kgUnitconfDisplayToREAL := Display / 0.03937;
			ELSE
				kgUnitconfDisplayToREAL := Display * 10;
			END_IF

		22:
			// mm dm inch
			IF LocUnit = KG_UNIT_US THEN
				kgUnitconfDisplayToREAL := Display / 0.03937;
			ELSE
				kgUnitconfDisplayToREAL := Display * 100;
			END_IF

		23:
			// mm m feet
			IF LocUnit = KG_UNIT_US THEN
				kgUnitconfDisplayToREAL := Display / 0.00328;
			ELSE
				kgUnitconfDisplayToREAL := Display * 1000;
			END_IF

		30:
			// 0,1kg kg lbs
			IF LocUnit = KG_UNIT_US THEN
				kgUnitconfDisplayToREAL := Display / 0.220462;
			ELSE
				kgUnitconfDisplayToREAL := Display * 10;
			END_IF

		40:
			// 0,1 °C °C °F
			IF LocUnit = KG_UNIT_US THEN
				kgUnitconfDisplayToREAL := (Display - 32.0) / 0.18;
			ELSE
				kgUnitconfDisplayToREAL := Display * 10;
			END_IF

		41:
			// °C °C °F
			IF LocUnit = KG_UNIT_US THEN
				kgUnitconfDisplayToREAL := (Display - 32.0) / 1.8;
			ELSE
				kgUnitconfDisplayToREAL := Display;
			END_IF

		50:
			// 0,1 bar bar psi
			IF LocUnit = KG_UNIT_US THEN
				kgUnitconfDisplayToREAL := Display / 1.450368;
			ELSE
				kgUnitconfDisplayToREAL := Display * 10;
			END_IF

		310:
			// 0,01 l/kg l/kg gal/lbs
			IF LocUnit = KG_UNIT_US THEN
				kgUnitconfDisplayToREAL := Display / 0.00119827;
			ELSE
				kgUnitconfDisplayToREAL := Display * 100;
			END_IF

		ELSE

			kgUnitconfDisplayToREAL := Display;

	END_CASE

END_FUNCTION
```

#### kgGetProgdata.st - Read Programdata from a dataobject
```iecst
(********************************************************************
 * COPYRIGHT -- Herbert Kannegiesser GmbH
 ********************************************************************
 * Library: KGstdLib
 * File: kgGetProgdata.st
 * Author: hunholz
 * Created: April 11, 2012
 ********************************************************************
 * Implementation of library KGstdLib
 ********************************************************************)

(* Read Programdata from a dataobject *)
FUNCTION kgGetProgdata

	IF LEN(sBaseName) = 0 THEN
		kgGetProgdata := KG_ERR_NULLSTRING;
		RETURN;
	END_IF

	IF pMem = 0 THEN
		kgGetProgdata := KG_ERR_NULPOINTER;
		RETURN;
	END_IF

	_sIndex := '';
	IF wProgMaxNo > 9999 AND  wProgNo  < 10000 THEN
		_sIndex := CONCAT(_sIndex,'0');
	END_IF
	IF wProgMaxNo > 999 AND  wProgNo  < 1000 THEN
		_sIndex := CONCAT(_sIndex,'0');
	END_IF
	IF wProgMaxNo > 99 AND  wProgNo  < 100 THEN
		_sIndex := CONCAT(_sIndex,'0');
	END_IF
	IF wProgMaxNo > 9 AND  wProgNo  < 10 THEN
		_sIndex := CONCAT(_sIndex,'0');
	END_IF

	_sIndex1 := UINT_TO_STRING(wProgNo);

	_sIndex := CONCAT(_sIndex, _sIndex1);

	_sName := CONCAT(sBaseName, _sIndex);

	_diProg(enable := TRUE, pName := ADR(_sName));

	IF _diProg.status = ERR_OK THEN

		IF _diProg.len > lSize THEN
			kgGetProgdata := KG_ERR_WRONGSIZES;
			RETURN;
		END_IF

		brsmemcpy(pMem, _diProg.pDatObjMem, _diProg.len);

		kgGetProgdata := ERR_OK;

		RETURN;

	ELSE
		kgGetProgdata := _diProg.status;
		RETURN;
	END_IF

END_FUNCTION
```

### KGStandard-History.txt
```
1.00.0	30.06.2011 NEU
1.01.0	02.07.2011 mnCnt ergänzt
1.02.0	08.07.2011 Netlink 1.02.0
1.03.0  19.07.2011 kgStd 1.01.0
1.04.0	26.07.2011 Maschinentyp in der Infostruktur auf 11 Zeichen verringert
1.05.0		   Keine Ahnung
1.06.0	01.09.2011 Info_typ erweitert
1.07.0	20.09.2011 Stat_typ ergänzt
1.08.0	06.10.2011 Netlink 1.05.0
1.08.1	14.10.2011 Netlink 1.06.0
1.09.0  03.11.2011 Umstellung auf AS 3.0.90
					- Stat_typ erweitert
					- Funktionen zum Generieren einer Postennummer in KGstdLib ergänzt 1.02.0
1.10.0	20.12.2011 Ringbufferfunktionen ergänzt
				   KGBOM ergänzt
				   KG_DEVICE_COMPACTFLASH ergänzt
1.11.0	03.01.2012 kgGUIDisZero : Funktion prüft, ob eine GUID null ist.
1.12.0	12.01.2012 kgNextBatchNoLong merkt sich die letzte Postennummer. BatchNo ist nur noch Output.
1.13.0	24.01.2012 Erweiterung der Ringbuffer-Funktionen. Einführung des Startzeigers.
				   Unabhängigkeit von Netlink. Netlink entfernt.
				   Konstanten für Maschinenstati ergänzt
				   Maschinentypen aus NetLink-Library übernommen. nlMachinetypeW3_typ --> kgMachinetypeW3_typ
				   Datentypen utfName15 und utfName31 als abgeleiteten Datentyp deklariert
1.14.0	03.02.2012 Im Pkg_KGStandardShare werden die Konstanten KG_DEVICE_USBSTICK1 und KG_DEVICE_USBSTICK2 als STRING[31] deklariert.
				   In der sysconf sollten die Device-Namen für gültige USB-Massenspeicher definiert sein.
1.15.0	08.02.2012 Funktionen: kgGetLineNumberW3 und kgGetMachineAdressW3. (mnEth Version 2.08.0 verwenden)
1.15.1	15.02.2012 kgGetBatchNoUnique und kgNextBatchNoLong korrigiert
1.16.0	15.03.2012 Konvertierung von Parametern entsprechend der Einheit (units.csv 2011-11-25T08:56:00)
1.16.1	15.03.2012 Für Displaywerte werden auch die Nachkommastellen mit angegeben
1.16.2	20.03.2012 Bugfix KGstdLib
1.17.0	21.03.2012 KGstdLib erweitert
1.17.1	22.03.2012 CP3585 ergänzt
1.18.0	04.04.2012 _Info_ gibt es nicht mehr
1.19.0	11.04.2012 Enumeration für Maschinenstati
```

### Package Logical/Mewa/KGFramework/Pkg_mnSystem - Systemtask für Versionierung

### Program Logical/Mewa/KGFramework/Pkg_mnSystem/mnSystem (IEC) - Systemtask für Versionierung

#### mnSystemCyclic.st - Cyclic code
```iecst
(********************************************************************
 * COPYRIGHT -- Kannegiesser GmbH
 ********************************************************************
 * Program: mnSystem
 * File: mnSystemCyclic.st
 * Author: Hunholz
 * Created: Mar 16, 2012
 ********************************************************************
 * Implementation of program mnSystem
 ********************************************************************)

PROGRAM _CYCLIC

	//**********************
	// USB Knoten überwachen
	//**********************

	// Alle 5 Sekunden eine Liste der verfügbaren Sticks zur Verfügung stellen

	_TONsearchForUSB(IN := _wUSBstate = 0 , PT := T#5s);

	CASE _wUSBstate OF

		0:

			IFmnSystem.Out.sInterfaceUSB := _sInterfaceUSB;
			IFmnSystem.Out.xUSBStickReady := _xUSBStickReady;

			IF _TONsearchForUSB.Q THEN

				_wUSBstate := 1;

			END_IF

		1:
			_UsbNodeListGet(enable := TRUE, pBuffer := ADR(_lUSBlist), bufferSize := SIZEOF(_lUSBlist), filterInterfaceClass := asusb_CLASS_MASS_STORAGE, filterInterfaceSubClass := asusb_SUBCLASS_SCSI_COMMAND_SET);

			IF _UsbNodeListGet.status <> ERR_FUB_BUSY THEN

				_sInterfaceUSB := '';
				_xUSBStickReady := FALSE;

				IF _UsbNodeListGet.status = ERR_OK THEN

					_wUSBstate := 2;

				ELSE

					_wUSBstate := 0;

				END_IF

			END_IF

		2:

			_UsbNodeGet(enable := TRUE, nodeId := _lUSBlist[1], pBuffer := ADR(_usbNode), bufferSize := SIZEOF(_usbNode));

			IF _UsbNodeGet.status <> ERR_FUB_BUSY THEN

				IF _UsbNodeGet.status = ERR_OK THEN

					brsmemcpy(ADR(_sInterfaceUSB),ADR(_usbNode.ifName),SIZEOF(_sInterfaceUSB));;
					_xUSBStickReady := TRUE;

				END_IF

				_wUSBstate := 0;

			END_IF

		ELSE

			_wUSBstate := 0;

	END_CASE

	//#####################################################################################################################

	// Heartbeeat erzeugen (Sekunden)
	_GetTime(enable := TRUE);
	mnSystemStatAd.wHeartbeat := DT_TO_UINT(_GetTime.DT1);

	// Lüfterüberwachung

	CASE IFmnSystem.In.PLC.wMDL_ID OF

		KG_CPU_X20CP1486:

			_xFanOk := IFmnSystem.In.PLC.xFanOk;

		ELSE

			_xFanOk := TRUE;

	END_CASE

	// Überwachung Umgebungstemperatur

	_TONtemp(IN := (IFmnSystem.In.PLC.wTemperatureENV > mnSystemPar.Mac.wWarnTemperatureEnvironment), PT := T#10m);

	// Meldungen
	IF NOT IFmnTest.Out.xNoMessages THEN

		kgMsgStatus[MNSYSTEM_IDX_KGMSGSTAT].wFunction_ID 	:= 110;

		IF NOT _xFanOk THEN

			kgMsgStatus[MNSYSTEM_IDX_KGMSGSTAT].wMsgClass		:= MNMSG_CLASS_WARNING;
			kgMsgStatus[MNSYSTEM_IDX_KGMSGSTAT].wMsgAckLevel	:= 0;
			kgMsgStatus[MNSYSTEM_IDX_KGMSGSTAT].wMsgNumber		:= MNSYSTEM_MSG_FAN;

		ELSIF _TONtemp.Q THEN

			kgMsgStatus[MNSYSTEM_IDX_KGMSGSTAT].wMsgClass		:= MNMSG_CLASS_WARNING;
			kgMsgStatus[MNSYSTEM_IDX_KGMSGSTAT].wMsgAckLevel	:= 0;
			kgMsgStatus[MNSYSTEM_IDX_KGMSGSTAT].wMsgNumber		:= MNSYSTEM_MSG_ENVTEMP;

		ELSIF IFmnSystem.In.PLC.bBatteryStatusCPU <> 1 THEN

			kgMsgStatus[MNSYSTEM_IDX_KGMSGSTAT].wMsgClass		:= MNMSG_CLASS_WARNING;
			kgMsgStatus[MNSYSTEM_IDX_KGMSGSTAT].wMsgAckLevel	:= 0;
			kgMsgStatus[MNSYSTEM_IDX_KGMSGSTAT].wMsgNumber		:= MNSYSTEM_MSG_BATTERY;

		ELSE

			kgMsgStatus[MNSYSTEM_IDX_KGMSGSTAT].wFunction_ID 	:= 110;
			kgMsgStatus[MNSYSTEM_IDX_KGMSGSTAT].wMsgClass		:= 0;
			kgMsgStatus[MNSYSTEM_IDX_KGMSGSTAT].wMsgAckLevel	:= 0;
			kgMsgStatus[MNSYSTEM_IDX_KGMSGSTAT].wMsgNumber		:= 0;

		END_IF

	END_IF

	// Stati
	mnSystemStatAd.lSerialNumber 			:= IFmnSystem.In.PLC.lSerialNumber;
	mnSystemStatAd.wTemperatureCPU 			:= IFmnSystem.In.PLC.wTemperatureCPU;
	mnSystemStatAd.wTemperatureEnvironment 	:= IFmnSystem.In.PLC.wTemperatureENV;

END_PROGRAM
```

#### mnSystemInit.st - Initialization code
```iecst
(********************************************************************
 * COPYRIGHT -- Kannegiesser GmbH
 ********************************************************************
 * Program: mnSystem
 * File: mnSystemInit.st
 * Author: horn
 * Created: January 10, 2012
 ********************************************************************
 * Implementation of program mnSystem
 ********************************************************************)

PROGRAM _INIT

	// Packet-Version auslesen mit MO_ver aus SYS_lib und für den Additional Status zur Verfügung stellen

	_sPkgName := 'mnSystem';

	IF ( MO_ver(ADR(_sPkgName), 0, ADR(_VerStruc)) = 0 ) THEN

		brsmemcpy(ADR(mnSystemStatAd.sPkgVersion), ADR(_VerStruc.version), SIZEOF(_VerStruc.version));

	ELSE

		mnSystemStatAd.sPkgVersion := '---';

	END_IF

	_sPkgName := 'mnMaster';

	IF ( MO_ver(ADR(_sPkgName), 0, ADR(_VerStruc)) = 0 ) THEN

		brsmemcpy(ADR(mnSystemStatAd.sPrjVersion), ADR(_VerStruc.version), SIZEOF(_VerStruc.version));

	ELSE

		mnSystemStatAd.sPrjVersion := '---';

	END_IF

	// CPU-Typ bestimmen

	CASE IFmnSystem.In.PLC.wMDL_ID OF

		KG_CPU_CTT_11:

			mnSystemStatAd.sCPUType := 'CTT-11';

		KG_CPU_PCT_03:

			mnSystemStatAd.sCPUType := 'PCT-03';

		KG_CPU_PCT_04:

			mnSystemStatAd.sCPUType := 'PCT-04';

		KG_CPU_PP65_0571_P74:

			mnSystemStatAd.sCPUType := 'PP65.0571.P74';

		KG_CPU_PP420_1043_75:

			mnSystemStatAd.sCPUType := 'PP420.1043.75';

		KG_CPU_X20CP1484:

			mnSystemStatAd.sCPUType := 'CP1484';

		KG_CPU_X20CP1484_1:

			mnSystemStatAd.sCPUType := 'CP1484-1';

		KG_CPU_X20CP1486:

			mnSystemStatAd.sCPUType := 'CP1486';

		KG_CPU_X20CP3484_1:

			mnSystemStatAd.sCPUType := 'CP3484-1';

		KG_CPU_X20CP3486:

			mnSystemStatAd.sCPUType := 'CP3486';

		KG_CPU_X20CP3585:

			mnSystemStatAd.sCPUType := 'CP3585';

		ELSE

			mnSystemStatAd.sCPUType := UINT_TO_STRING(IFmnSystem.In.PLC.wMDL_ID);

	END_CASE

	_wMdlId := IFmnSystem.In.PLC.wMDL_ID;

END_PROGRAM
```

#### _mnSystem.var - Local variables
```iecst
(********************************************************************
 * COPYRIGHT -- Kannegiesser GmbH
 ********************************************************************
 * Program: mnSystem
 * File: _mnSystem.var
 * Author: horn
 * Created: January 10, 2012
 ********************************************************************
 * Local variables of program mnSystem
 ********************************************************************)
VAR
	_sPkgName : STRING[11];
	_VerStruc : MoVerStruc_typ;
	_GetTime : DTGetTime;
	_xFanOk : BOOL;
	_wMdlId : UINT;
	_TONtemp : TON;
	_wUSBstate : UINT;
	_TONsearchForUSB : TON;
	_lUSBlist : ARRAY[1..3] OF UDINT;
	_UsbNodeListGet : UsbNodeListGet;
	_sInterfaceUSB : STRING[31];
	_xUSBStickReady : BOOL;
	_lAttachDetachCount : UDINT;
	_usbNode : usbNode_typ;
	_UsbNodeGet : UsbNodeGet;
END_VAR
```

### mnSystem.typ - Local data types
```iecst
(********************************************************************
 * COPYRIGHT -- Kannegiesser GmbH
 ********************************************************************
 * Program: mnSystem
 * File: mnSystem.typ
 * Author: horn
 * Created: January 10, 2012
 ********************************************************************
 * Local data types of program mnSystem
 ********************************************************************)

TYPE
	mnSystemStatAd_typ : 	STRUCT
		sPkgVersion : STRING[10]; (*Version des Packes mnSystem*)
		sPrjVersion : STRING[10]; (*Hauptversion des Projektes*)
		sCPUType : STRING[19]; (*CPU-Typ*)
		wHeartbeat : UINT; (*Zählt sekündlich hoch*)
		wTemperatureCPU : UINT; (*CPU Temperatur 1/10 °C*)
		wTemperatureEnvironment : UINT; (*Umgebungstemperatur 1/10 °C*)
		lSerialNumber : UDINT; (*Seriennummer der CPU*)
	END_STRUCT;
	IFmnSystem_typ : 	STRUCT
		In : IFmnSystemIn_typ;
		Out : IFmnSystemOut_typ;
	END_STRUCT;
	IFmnSystemOut_typ : 	STRUCT
		xUSBStickReady : BOOL; (*USB-Stick erkannt*)
		sInterfaceUSB : STRING[31]; (*Interfacebezeichnung für den Stick*)
	END_STRUCT;
	IFmnSystemIn_typ : 	STRUCT
		PLC : mnSystem_PLC_typ;
	END_STRUCT;
	mnSystem_PLC_typ : 	STRUCT
		lSerialNumber : UDINT; (*Serien-Nummer des X20 Moduls*)
		wMDL_ID : UINT; (*Modul-ID des X20 Moduls*)
		bModeSwitch : USINT; (*Version der Firmware*)
		bBatteryStatusCPU : USINT; (*Status der Pufferbatterie*)
		xFanOk : BOOL; (*Status des CPU-Lüfters*)
		wTemperatureCPU : UINT; (*CPU-Temperatur*)
		wTemperatureENV : UINT;
		diSystemTime : DINT; (*Systemzeit der CPU in µs*)
		xStatusInput01 : BOOL; (*Status der 24V-Versorgung für I/O*)
	END_STRUCT;
	mnSystemPar_typ : 	STRUCT
		Mac : mnSystemParMac_typ;
	END_STRUCT;
	mnSystemParMac_typ : 	STRUCT
		wWarnTemperatureEnvironment : UINT := 750; (*Warnschwelle für Temperaturüberwachung in 0,1 °C*)
	END_STRUCT;
END_TYPE
```

### mnSystem.var - Local variables
```iecst
(********************************************************************
 * COPYRIGHT -- Kannegiesser GmbH
 ********************************************************************
 * Program: mnSystem
 * File: mnSystem.var
 * Author: horn
 * Created: January 10, 2012
 ********************************************************************
 * Local variables of program mnSystem
 ********************************************************************)
(*Konstanten*)
VAR CONSTANT
	MNSYSTEM_MSG_BATTERY : UINT := 3;
	MNSYSTEM_MSG_FAN : UINT := 4;
	MNSYSTEM_MSG_ENVTEMP : UINT := 5;
END_VAR
(*Variablen*)
VAR
	IFmnSystem : IFmnSystem_typ;
	mnSystemCmd : KG_Cmd_typ;
	mnSystemStat : Stat_typ;
	mnSystemStatAd : mnSystemStatAd_typ;
	mnSystemPar : mnSystemPar_typ;
END_VAR
```

### mnSystem.History.txt
```
1.00.0	2012-03-16	AH	Neu
1.00.1	2012-03-20 	AH	Abhängigkeiten ergänzt
1.01.0	2012-03-23	AH	Lüfterüberwachung, Temperaturüberwachung
1.02.0	2012-03-23	AH	USB-Stick Überwachung
1.02.1	2012-04-17	AH	Bei unbekannter Modul-ID wird die Modul-ID als CPU-Typ zurückgegeben.
```

### CfgMsgStat.mnSystem.txt
```
;****************************
; System Manager
;*****************************
00110, 00003, 00000, 00000;
00110, 00004, 00000, 00000;
00110, 00005, 00000, 00000;
```

### Package Logical/Mewa/KGFramework/Pkg_mnEth - Ethernet Manager

### Pkg_mnEth.typ - Global data types
```iecst
(********************************************************************
 * COPYRIGHT --
 ********************************************************************
 * File: Global.typ
 * Author: tamme
 * Created: March 17, 2011
 ********************************************************************
 * Global data types of project Ethernetmanagr
 ********************************************************************)

TYPE
	mnEthIP_typ : 	STRUCT
		sIP : STRING[15];
		sGateway : STRING[15];
		sHostname : STRING[15];
		sNetId : STRING[15];
		bNetId1 : USINT;
		bNetId2 : USINT;
		bNetId3 : USINT;
		bRegion : USINT;
		bStation : USINT;
		bNumber : USINT;
	END_STRUCT;
	IFmnEthOut_typ : 	STRUCT
		IP : mnEthIP_typ;
		xDataValid : BOOL;
	END_STRUCT;
	IFmnEth_typ : 	STRUCT
		Out : IFmnEthOut_typ;
	END_STRUCT;
	mnEthStatAd_typ : 	STRUCT
		IP : mnEthIP_typ;
		xDataValid : BOOL;
		sPkgVersion : STRING[11];
	END_STRUCT;
	mnEthPar_typ : 	STRUCT
		Cfg : mnEthParCfg_typ;
		Mac : mnEthParMac_typ;
	END_STRUCT;
	mnEthParMac_typ : 	STRUCT
		xStartDHCP : BOOL;
		xStartSNTPClt : BOOL;
		xStartSNTPSrv : BOOL;
		xReserve : USINT;
		sIP_SNTP_Srv : STRING[15];
	END_STRUCT;
	mnEthParCfg_typ : 	STRUCT
		bNETid1 : USINT;
		bNETid2 : USINT;
		bNETid3 : USINT;
		bRegion : USINT;
		bStation : USINT;
	END_STRUCT;
END_TYPE
```

### Program Logical/Mewa/KGFramework/Pkg_mnEth/mnEth (IEC) - Ethernetmanager

#### mnEthCyclic.st - Cyclic code
```iecst
(********************************************************************
 * COPYRIGHT --
 ********************************************************************
 * Program: mnEth
 * File: mnEthCyclic.st
 * Author: hunholz
 * Created: August 9, 2011
 * Changed: October 7, 2011
 ********************************************************************
 * Implementation of program mnEth
 ********************************************************************)

PROGRAM _CYCLIC

	// Input Messagesystem

	_kgMsgStatus.xAckAva := kgMsgStatus[MNETH_IDX_KGMSGSTAT].xAckAva;
	_kgMsgStatus.xAckFault := kgMsgStatus[MNETH_IDX_KGMSGSTAT].xAckFault;
	_kgMsgStatus.xAckMaint := kgMsgStatus[MNETH_IDX_KGMSGSTAT].xAckMaint;

	_kgMsgStatus.wFunction_ID := 4;

	IF _xmnEthOk THEN

		CASE enEState OF

			es_idle:

				IF _xSetHostname THEN

					enEState := es_SetHostname1;

				ELSIF _xSetDefault THEN

					enEState := es_SetDef1;

				ELSIF mnEthPar.Mac.xStartDHCP AND IFmnParam.Out.xParamOK AND NOT _xDHCPstarted THEN

					// schaltet den DHCP-Server ein. Nicht dauerhaft. Wird der Maschinenparameter auf FALSE gesetzt
					// dann bleibt der DHCP-Server aus.
					enEState := es_DHCP1;

				ELSIF mnEthPar.Mac.xStartSNTPClt AND IFmnParam.Out.xParamOK AND NOT _xSNTPCltStarted THEN

					enEState := es_SNTPcltStart1;

				ELSIF NOT mnEthPar.Mac.xStartSNTPClt AND IFmnParam.Out.xParamOK AND _xSNTPCltStarted THEN

					enEState := es_SNTPcltStop1;

				ELSIF mnEthPar.Mac.xStartSNTPSrv AND IFmnParam.Out.xParamOK AND NOT _xSNTPSrvStarted THEN

					enEState := es_SNTPsrvStart1;

				ELSIF NOT mnEthPar.Mac.xStartSNTPSrv AND IFmnParam.Out.xParamOK AND _xSNTPSrvStarted THEN

					enEState := es_SNTPsrvStop1;

				ELSIF _bWaitCounter >= 3 THEN

					_xChanged := FALSE;

					_ParSet := _ParAktuell;

					enEState := es_WriteCSV1;

				ELSIF _TONidle.Q THEN

					enEState := es_Change1;

				END_IF

			// Beobachte eingestellte IP und das Gateway
			es_Change1:

				_CfgGetGateway(enable := TRUE, pDevice := ADR(_sEthDevice), pGateway := ADR(_ParGet.Gateway_Adr), Len := SIZEOF(_ParGet.Gateway_Adr));

				IF _CfgGetGateway.status = ERR_OK THEN

					enEState := es_Change2;

				ELSIF _CfgGetGateway.status <> ERR_FUB_BUSY THEN

					_kgMsgStatus.wMsgClass := 11;
					_kgMsgStatus.wMsgNumber := _MENETH_MSG_CHANGE;
					_kgMsgStatus.diMsgAttr1 := UINT_TO_DINT(_CfgGetGateway.status);

					enEState := es_Warning;
				END_IF

			es_Change2:

				_CfgGetIPAddress(enable := TRUE, pDevice := ADR(_sEthDevice), pIPAddr := ADR(_ParGet.IP_Adr), Len := SIZEOF(_ParGet.IP_Adr));

				IF _CfgGetIPAddress.status = ERR_OK THEN

					enEState := es_Change3;

				ELSIF _CfgGetIPAddress.status <> ERR_FUB_BUSY THEN

					_kgMsgStatus.wMsgClass := 11;
					_kgMsgStatus.wMsgNumber := _MENETH_MSG_CHANGE;
					_kgMsgStatus.diMsgAttr1 := UINT_TO_DINT(_CfgGetIPAddress.status);

					enEState := es_Warning;
				END_IF

			es_Change3:

				IF (brsstrcmp(ADR(_ParAktuell.Gateway_Adr), ADR(_ParGet.Gateway_Adr)) = 0)	AND (brsstrcmp(ADR(_ParAktuell.IP_Adr), ADR(_ParGet.IP_Adr)) = 0) THEN

					IF _xChanged THEN

						_bWaitCounter := _bWaitCounter + 1;

					ELSE

						_bWaitCounter := 0;

					END_IF

					enEState := es_idle;

				ELSE

					IF ethInetAton(pIpStr := ADR(_ParGet.IP_Adr), ADR(_lIPAdr)) = ERR_OK THEN

						IF ethInetAton(pIpStr := ADR(_ParGet.Gateway_Adr), ADR(_lGatewayAdr)) = ERR_OK THEN

							_pOctet ACCESS ADR(_lIPAdr);

							_ParGet.IP_ID1 := _pOctet[0];
							_ParGet.IP_ID2 := _pOctet[1];
							_ParGet.IP_ID3 := (_pOctet[2] / 16) * 16;
							_ParGet.Region := _pOctet[2] MOD 16;
							_ParGet.Station := _pOctet[3];

							IF _ParGet.Region = 3 THEN
								_ParGet.Number := kgGetLineNumberW3(Station := _ParGet.Station, pMachineType := ADR(_kgMachineTypeW3));
							ELSE
								_ParGet.Number := 0;
							END_IF

							// NET-Id bestimmen
							_lNetId := _lIPAdr;
							_pOctet ACCESS ADR(_lNetId);

							_pOctet[2] := _ParGet.IP_ID3;
							_pOctet[3] := 0;

							ethInetNtoa(ipAdr := _lNetId, pIpStr := ADR(_ParGet.NetId_Adr));

							_pOctet ACCESS ADR(_lGatewayAdr);

							_ParGet.GW_ID1 := _pOctet[0];
							_ParGet.GW_ID2 := _pOctet[1];
							_ParGet.GW_ID3 := _pOctet[2];
							_ParGet.GW_ID4 := _pOctet[3];

							enEState := es_Change4;

						END_IF

					END_IF

				END_IF

			es_Change4:

				_CfgSetIPAddr(enable := TRUE, pDevice := ADR(_sEthDevice), pIPAddr := ADR(_ParGet.IP_Adr), Option := cfgOPTION_NON_VOLATILE);

				IF _CfgSetIPAddr.status = ERR_OK THEN

					enEState := es_Change5;

				ELSIF _CfgSetIPAddr.status <> ERR_FUB_BUSY THEN

					_kgMsgStatus.wMsgClass := 11;
					_kgMsgStatus.wMsgNumber := _MENETH_MSG_CHANGE;
					_kgMsgStatus.diMsgAttr1 := UINT_TO_DINT(_CfgSetIPAddr.status);

					enEState := es_Warning;

				END_IF

			es_Change5:

				_CfgSetDefaultGateway(enable := TRUE, pDevice := ADR(_sEthDevice), pGateway := ADR(_ParGet.Gateway_Adr), Option := cfgOPTION_NON_VOLATILE);

				IF _CfgSetDefaultGateway.status = ERR_OK THEN

					enEState := es_Change6;

				ELSIF _CfgSetDefaultGateway.status <> ERR_FUB_BUSY THEN

					_kgMsgStatus.wMsgClass := 11;
					_kgMsgStatus.wMsgNumber := _MENETH_MSG_CHANGE;
					_kgMsgStatus.diMsgAttr1 := UINT_TO_DINT(_CfgSetDefaultGateway.status);

					enEState := es_Warning;

				END_IF

			es_Change6:

// Für Testzwecke in Hausnetzen mit anderer Netzwerkmaske

#ifndef NoSubnetMask

				_CfgSetSubnetMask(enable := TRUE, pDevice := ADR(_sEthDevice), pSubnetMask := ADR(_sSubnetMask), Option := cfgOPTION_NON_VOLATILE);

				IF _CfgSetSubnetMask.status <> ERR_FUB_BUSY THEN

					enEState := es_Change7;

				END_IF
#else

				enEState := es_Change7;

#endif

			es_Change7:

				_pOctet ACCESS ADR(_lBroadcastAdr);

				_pOctet[0] := _ParGet.IP_ID1;
				_pOctet[1] := _ParGet.IP_ID2;
				_pOctet[2] := _ParGet.IP_ID3 + 15;
				_pOctet[3] := 255;

				ethInetNtoa(ADR(_lBroadcastAdr), ADR(_sBroadcastAdr));

				_CfgSetBroadcastAdr(enable := TRUE, pDevice := ADR(_sEthDevice), pBroadcastAddr := ADR(_sBroadcastAdr), Option := cfgOPTION_NON_VOLATILE);

				IF _CfgSetBroadcastAdr.status = ERR_OK THEN

					_ParAktuell := _ParGet;

					_xChanged  := TRUE;

					enEState := es_idle;

				ELSIF _CfgSetBroadcastAdr.status <> ERR_FUB_BUSY THEN

					_kgMsgStatus.wMsgClass := 11;
					_kgMsgStatus.wMsgNumber := _MENETH_MSG_SETDEF;
					_kgMsgStatus.diMsgAttr1 := UINT_TO_DINT(_CfgSetBroadcastAdr.status);

					enEState := es_Warning;

				END_IF

			// Setze Default aus Parameter
			es_SetDef1:

				IF IFmnParam.Out.xParamOK THEN

					_ParSet.IP_ID1 := mnEthPar.Cfg.bNETid1;
					_ParSet.IP_ID2 := mnEthPar.Cfg.bNETid2;
					_ParSet.IP_ID3 := mnEthPar.Cfg.bNETid3;
					_ParSet.Region := mnEthPar.Cfg.bRegion;
					_ParSet.Station := mnEthPar.Cfg.bStation;

					IF _ParAktuell.Region = 3 THEN
						_ParSet.Number := kgGetLineNumberW3(Station := _ParSet.Station, pMachineType := ADR(_kgMachineTypeW3));
					ELSE
						_ParSet.Number := 0;
					END_IF

					_pOctet ACCESS ADR(_lIPAdr);

					_pOctet[0] := _ParSet.IP_ID1;
					_pOctet[1] := _ParSet.IP_ID2;
					_pOctet[2] := _ParSet.IP_ID3 + _ParSet.Region;
					_pOctet[3] := _ParSet.Station;

					ethInetNtoa(_lIPAdr, ADR(_ParSet.IP_Adr));

					// NET-Id bestimmen
					_lNetId := _lIPAdr;
					_pOctet ACCESS ADR(_lNetId);

					_pOctet[2] := _ParSet.IP_ID3;
					_pOctet[3] := 0;

					ethInetNtoa(ipAdr := _lNetId, pIpStr := ADR(_ParSet.NetId_Adr));

					enEState := es_SetDef2;

				END_IF

			es_SetDef2:

				_CfgSetIPAddr(enable := TRUE, pDevice := ADR(_sEthDevice), pIPAddr := ADR(_ParSet.IP_Adr), Option := cfgOPTION_VOLATILE);

				IF _CfgSetIPAddr.status = ERR_OK THEN

					enEState := es_SetDef3;

				ELSIF _CfgSetIPAddr.status <> ERR_FUB_BUSY THEN

					_kgMsgStatus.wMsgClass := 11;
					_kgMsgStatus.wMsgNumber := _MENETH_MSG_SETDEF;
					_kgMsgStatus.diMsgAttr1 := UINT_TO_DINT(_CfgSetIPAddr.status);

					_xSetDefault := FALSE;
					enEState := es_Warning;

				END_IF

			es_SetDef3:

				_CfgGetGateway(enable := TRUE, pDevice := ADR(_sEthDevice), pGateway := ADR(_ParSet.Gateway_Adr), Len := SIZEOF(_ParSet.Gateway_Adr));

				IF _CfgGetGateway.status = ERR_OK THEN

					enEState := es_SetDef4;

				ELSIF _CfgGetGateway.status <> ERR_FUB_BUSY THEN

					_kgMsgStatus.wMsgClass := 11;
					_kgMsgStatus.wMsgNumber := _MENETH_MSG_SETDEF;
					_kgMsgStatus.diMsgAttr1 := UINT_TO_DINT(_CfgGetGateway.status);

					_xSetDefault := FALSE;
					enEState := es_Warning;

				END_IF

			es_SetDef4:

// Für Testzwecke in Hausnetzen mit anderer Netzwerkmaske

#ifndef NoSubnetMask

				_CfgSetSubnetMask(enable := TRUE, pDevice := ADR(_sEthDevice), pSubnetMask := ADR(_sSubnetMask), Option := cfgOPTION_VOLATILE);

				IF _CfgSetSubnetMask.status <> ERR_FUB_BUSY THEN

					enEState := es_SetDef5;

				END_IF
#else

				enEState := es_SetDef5;

#endif

			es_SetDef5:

				_pOctet ACCESS ADR(_lBroadcastAdr);

				_pOctet[0] := _ParSet.IP_ID1;
				_pOctet[1] := _ParSet.IP_ID2;
				_pOctet[2] := _ParSet.IP_ID3 + 15;
				_pOctet[3] := 255;

				ethInetNtoa(ADR(_lBroadcastAdr), ADR(_sBroadcastAdr));

				_CfgSetBroadcastAdr(enable := TRUE, pDevice := ADR(_sEthDevice), pBroadcastAddr := ADR(_sBroadcastAdr), Option := cfgOPTION_VOLATILE);

				IF _CfgSetBroadcastAdr.status = ERR_OK THEN

					_xSetDefault := FALSE;
					enEState := es_WriteCSV1;

				ELSIF _CfgSetBroadcastAdr.status <> ERR_FUB_BUSY THEN

					_kgMsgStatus.wMsgClass := 11;
					_kgMsgStatus.wMsgNumber := _MENETH_MSG_SETDEF;
					_kgMsgStatus.diMsgAttr1 := UINT_TO_DINT(_CfgSetBroadcastAdr.status);

					_xSetDefault := FALSE;
					enEState := es_Warning;

				END_IF

			es_WriteCSV1:

				_ParAktuell := _ParSet;

				brsmemset(_pParseMem, 0, 256);

				_lFileSize := 0;

				brwcsconv(ADR( _IPRow.utfIP_Adress), ADR(_ParSet.IP_Adr), 0);
				brwcsconv(ADR(_IPRow.utfGateway), ADR(_ParSet.Gateway_Adr), 0);

				_WriteBOM(enable := TRUE, pMem := _pParseMem, lMaxSize := 256, lSize := _lFileSize);
				_WriteCsv90(enable := TRUE, pMem := _pParseMem, lMaxSize := 256, IPRow := _IPRow, lSize := _lFileSize);

				enEState := es_WriteCSV2;

			es_WriteCSV2:

				_FileDeleteCsv(enable := TRUE, pDevice := ADR(KG_DEVICE_COMPACTFLASH), pName := ADR(_sPathCsv));

				IF _FileDeleteCsv.status <> ERR_FUB_BUSY THEN

					enEState := es_WriteCSV3;

				END_IF

			es_WriteCSV3:

				_FileCreateCsv(enable := TRUE, pDevice := ADR(KG_DEVICE_COMPACTFLASH), pFile := ADR(_sPathCsv));

				IF _FileCreateCsv.status = ERR_OK THEN

					enEState := es_WriteCSV4;

				ELSIF _FileCreateCsv.status <> ERR_FUB_BUSY THEN

					_kgMsgStatus.wMsgClass := 11;
					_kgMsgStatus.wMsgNumber := _MENETH_MSG_WRITECSV;
					_kgMsgStatus.diMsgAttr1 := UINT_TO_DINT(_FileCreateCsv.status);

					enEState := es_Warning;

				END_IF

			es_WriteCSV4:

				_FileOpenCsv(enable := TRUE, pDevice := ADR(KG_DEVICE_COMPACTFLASH), pFile := ADR(_sPathCsv), mode := fiWRITE_ONLY);

				IF _FileOpenCsv.status = ERR_OK THEN

					enEState := es_WriteCSV5;

				ELSIF _FileOpenCsv.status <> ERR_FUB_BUSY THEN

					_kgMsgStatus.wMsgClass := 11;
					_kgMsgStatus.wMsgNumber := _MENETH_MSG_WRITECSV;
					_kgMsgStatus.diMsgAttr1 := UINT_TO_DINT(_FileOpenCsv.status);

					enEState := es_Warning;

				END_IF

			es_WriteCSV5:

				_FileWriteCsv(enable := TRUE, ident := _FileOpenCsv.ident, offset := 0, pSrc := _pParseMem, len := _lFileSize);

				IF _FileWriteCsv.status <> ERR_FUB_BUSY THEN

					enEState := es_WriteCSV6;

				END_IF

			es_WriteCSV6:

				_FileCloseCsv(enable := TRUE, ident := _FileOpenCsv.ident);

				IF _FileCloseCsv.status <> ERR_FUB_BUSY THEN

					_bWaitCounter := 0;
					_xChanged := FALSE;

					enEState := es_idle;

				END_IF

			es_Warning:

				_bWaitCounter := 0;
				_xChanged := FALSE;

				IF _TONwarning.Q THEN

					brsmemset(ADR(_kgMsgStatus),0,SIZEOF(kgMsgStatus[0]));
					_kgMsgStatus.wFunction_ID := 4;

					enEState := es_idle;

				END_IF

			es_DHCP1:

				brsstrcpy(ADR(_cfgLease.name), ADR('KANLINK'));
				brsstrcpy(ADR(_cfgLease.defaultGateway), ADR(_ParAktuell.Gateway_Adr));
				brsstrcpy(ADR(_cfgLease.subnetMask), ADR(_sSubnetMask));

				// Startadresse
				_lIPAdr := 0;
				_pOctet ACCESS ADR(_lIPAdr);
				_pOctet[0] := _ParAktuell.IP_ID1;
				_pOctet[1] := _ParAktuell.IP_ID2;
				_pOctet[2] := _ParAktuell.IP_ID3;

				_pOctet[3] := 150;

				ethInetNtoa(_lIPAdr, ADR(_cfgLease.startAdr));

				// Stopadresse
				_pOctet[3] := 169;

				ethInetNtoa(_lIPAdr, ADR(_cfgLease.stopAdr));

				_cfgLease.leaseTimeout := -1;

				enEState := es_DHCP2;

			es_DHCP2:

				_CfgSetDhcpsData(enable := TRUE, pInterfaceList := ADR(_sEthDevice), pLeases := ADR(_cfgLease), numLeases := 1, option := cfgOPTION_VOLATILE);

				IF (_CfgSetDhcpsData.status = ERR_OK) THEN

					enEState := es_DHCP3;

				ELSIF _CfgSetDhcpsData.status <> ERR_FUB_BUSY THEN

					enEState := es_idle;
					_xDHCPstarted := TRUE;

				END_IF

			es_DHCP3:

				_CfgSetDhcpServer(enable := TRUE, start := 1, option := cfgOPTION_VOLATILE);

				IF _CfgSetDhcpServer.status <> ERR_FUB_BUSY THEN

					enEState := es_idle;
					_xDHCPstarted := TRUE;

				END_IF

			es_SNTPcltStart1:

				_CfgSetSntpClient(enable := TRUE, run := 1, pServerAddr := ADR(mnEthPar.Mac.sIP_SNTP_Srv), sntpcInterval := 30, rtcInterval := 30, option := cfgOPTION_VOLATILE);

				IF _CfgSetSntpClient.status <> ERR_FUB_BUSY THEN

					enEState := es_idle;
					_xSNTPCltStarted := TRUE;

				END_IF

			es_SNTPcltStop1:

				_CfgSetSntpClient(enable := TRUE, run := 0, pServerAddr := ADR(mnEthPar.Mac.sIP_SNTP_Srv), sntpcInterval := 30, rtcInterval := 30, option := cfgOPTION_VOLATILE);

				IF _CfgSetSntpClient.status <> ERR_FUB_BUSY THEN

					enEState := es_idle;
					_xSNTPCltStarted := FALSE;

				END_IF

			es_SNTPsrvStart1:

				_CfgSetSntpServer(enable := TRUE, start := 1, option := cfgOPTION_VOLATILE);

				IF _CfgSetSntpServer.status <> ERR_FUB_BUSY THEN

					enEState := es_idle;
					_xSNTPSrvStarted := TRUE;

				END_IF

			es_SNTPsrvStop1:

				_CfgSetSntpServer(enable := TRUE, start := 0, option := cfgOPTION_VOLATILE);

				IF _CfgSetSntpServer.status <> ERR_FUB_BUSY THEN

					enEState := es_idle;
					_xSNTPSrvStarted := FALSE;

				END_IF

			es_SetHostname1:

				IF IFmnParam.Out.xParamOK THEN

					brwcsconv(ADR(_sMnr), ADR(IFmnParam.Out.utfMachineNumber) ,1);

					_sHostname := 'KaMa';
					brsstrcat(ADR(_sHostname), ADR(_sMnr));

					enEState := es_SetHostname2;

				END_IF

			es_SetHostname2:

				_CfgGetHostName(enable := TRUE, pHostName := ADR(_sActHostname), Len := SIZEOF(_sActHostname));

				IF _CfgGetHostName.status = ERR_OK THEN

					IF brsstrcmp(ADR(_sHostname), ADR(_sActHostname)) = 0 THEN

						_xSetHostname := FALSE;
						enEState := es_idle;

					ELSE

						enEState := es_SetHostname3;

					END_IF

				ELSIF _CfgGetHostName.status <> ERR_FUB_BUSY THEN

					_xSetHostname := FALSE;
					enEState := es_idle;

				END_IF

			es_SetHostname3:

				_CfgSetHostName(enable := TRUE, pHostName := ADR(_sHostname), Option := cfgOPTION_NON_VOLATILE);

				IF _CfgSetHostName.status <> ERR_FUB_BUSY THEN

					_xSetHostname := FALSE;
					enEState := es_idle;

				END_IF

		END_CASE

		_TONidle(IN := enEState = es_idle, PT := T#30s);

		_TONwarning(IN := enEState = es_Warning, PT := T#30s);

		// Ethernetdaten übergeben
		mnEthStatAd.IP.sHostname		:= _sHostname;
		mnEthStatAd.IP.sIP 				:= _ParAktuell.IP_Adr;
		mnEthStatAd.IP.sGateway 		:= _ParAktuell.Gateway_Adr;
		mnEthStatAd.IP.sNetId			:= _ParAktuell.NetId_Adr;
		mnEthStatAd.IP.bNetId1			:= _ParAktuell.IP_ID1;
		mnEthStatAd.IP.bNetId2			:= _ParAktuell.IP_ID2;
		mnEthStatAd.IP.bNetId3			:= _ParAktuell.IP_ID3;
		mnEthStatAd.IP.bNumber			:= _ParAktuell.Number;
		mnEthStatAd.IP.bRegion			:= _ParAktuell.Region;
		mnEthStatAd.IP.bStation			:= _ParAktuell.Station;
		IFmnEth.Out.IP					:= mnEthStatAd.IP;
		mnEthStatAd.xDataValid			:= NOT _xSetDefault AND NOT _xSetHostname;
		IFmnEth.Out.xDataValid			:= mnEthStatAd.xDataValid;

	ELSE

		_kgMsgStatus.wMsgClass := 11;

		mnEthStatAd.xDataValid := FALSE;

	END_IF // _xmnEthOk

	// MsgSystem Output

	IF NOT IFmnTest.Out.xNoMessages THEN

		kgMsgStatus[MNETH_IDX_KGMSGSTAT].diMaintAttr1 		:= _kgMsgStatus.diMaintAttr1;
		kgMsgStatus[MNETH_IDX_KGMSGSTAT].diMaintAttr2 		:= _kgMsgStatus.diMaintAttr2;
		kgMsgStatus[MNETH_IDX_KGMSGSTAT].diMsgAttr1 		:= _kgMsgStatus.diMsgAttr1;
		kgMsgStatus[MNETH_IDX_KGMSGSTAT].diMsgAttr2 		:= _kgMsgStatus.diMsgAttr2;
		kgMsgStatus[MNETH_IDX_KGMSGSTAT].sMaintAttrTxt 		:= _kgMsgStatus.sMaintAttrTxt;
		kgMsgStatus[MNETH_IDX_KGMSGSTAT].sMsgAttrTxt		:= _kgMsgStatus.sMsgAttrTxt;
		kgMsgStatus[MNETH_IDX_KGMSGSTAT].wFunction_ID		:= _kgMsgStatus.wFunction_ID;
		kgMsgStatus[MNETH_IDX_KGMSGSTAT].wInstance			:= _kgMsgStatus.wInstance;
		kgMsgStatus[MNETH_IDX_KGMSGSTAT].wMaintAckLevel		:= _kgMsgStatus.wMaintAckLevel;
		kgMsgStatus[MNETH_IDX_KGMSGSTAT].wMaintNumber		:= _kgMsgStatus.wMaintNumber;
		kgMsgStatus[MNETH_IDX_KGMSGSTAT].wMsgAckLevel		:= _kgMsgStatus.wMsgAckLevel;
		kgMsgStatus[MNETH_IDX_KGMSGSTAT].wMsgClass			:= _kgMsgStatus.wMsgClass;
		kgMsgStatus[MNETH_IDX_KGMSGSTAT].wMsgNumber			:= _kgMsgStatus.wMsgNumber;
		kgMsgStatus[MNETH_IDX_KGMSGSTAT].xAckRead			:= _kgMsgStatus.xAckRead;

	END_IF

END_PROGRAM
```
